	ARdsEventCtrl[314].bSignalInput							:=	NOT bChillerSystemTempHAL; //(* MAIN INC CHILLED WATER *):	 
	ARdsEventCtrl[314].iDelayTimeSV							:=	0;
	ARdsEventCtrl[314].bHoldingDisable;
	ARdsEventCtrl[314].bTest_InvertedInputEn;
	ARdsEventCtrl[314].bEventOutput;
	
	ARdsEventCtrl[315].bSignalInput							:=ARbStnTempPreparationNoRdyAlarm[1];// PROCESS TANK 1 TEMP PREPARATION NO READY ALARM 
	ARdsEventCtrl[315].iDelayTimeSV							:=0;
	ARdsEventCtrl[315].bHoldingDisable;
	ARdsEventCtrl[315].bTest_InvertedInputEn;
	ARdsEventCtrl[315].bEventOutput;

	
	ARdsEventCtrl[316].bSignalInput							:=ARbStnTempPreparationNoRdyAlarm[2];// PROCESS TANK 2 TEMP PREPARATION NO READY ALARM 
	ARdsEventCtrl[316].iDelayTimeSV							:=0;
	ARdsEventCtrl[316].bHoldingDisable;
	ARdsEventCtrl[316].bTest_InvertedInputEn;
	ARdsEventCtrl[316].bEventOutput;

	
	ARdsEventCtrl[317].bSignalInput							:=ARbStnTempPreparationNoRdyAlarm[3];// PROCESS TANK 3 TEMP PREPARATION NO READY ALARM 
	ARdsEventCtrl[317].iDelayTimeSV							:=0;
	ARdsEventCtrl[317].bHoldingDisable;
	ARdsEventCtrl[317].bTest_InvertedInputEn;
	ARdsEventCtrl[317].bEventOutput;

	
	ARdsEventCtrl[318].bSignalInput							:=ARbStnTempPreparationNoRdyAlarm[4];// PROCESS TANK 4 TEMP PREPARATION NO READY ALARM 
	ARdsEventCtrl[318].iDelayTimeSV							:=0;
	ARdsEventCtrl[318].bHoldingDisable;
	ARdsEventCtrl[318].bTest_InvertedInputEn;
	ARdsEventCtrl[318].bEventOutput;

	ARdsEventCtrl[319].bSignalInput							:=ARbStnTempPreparationNoRdyAlarm[5];// PROCESS TANK 5 TEMP PREPARATION NO READY ALARM 
	ARdsEventCtrl[319].iDelayTimeSV							:=0;
	ARdsEventCtrl[319].bHoldingDisable;
	ARdsEventCtrl[319].bTest_InvertedInputEn;
	ARdsEventCtrl[319].bEventOutput;
	
	ARdsEventCtrl[320].bSignalInput							:=ARbStnTempPreparationNoRdyAlarm[6];// PROCESS TANK 6 TEMP PREPARATION NO READY ALARM 
	ARdsEventCtrl[320].iDelayTimeSV							:=0;
	ARdsEventCtrl[320].bHoldingDisable;
	ARdsEventCtrl[320].bTest_InvertedInputEn;
	ARdsEventCtrl[320].bEventOutput;
	
	ARdsEventCtrl[321].bSignalInput							:=ARbStnTempPreparationNoRdyAlarm[7];// PROCESS TANK 7 TEMP PREPARATION NO READY ALARM  
	ARdsEventCtrl[321].iDelayTimeSV							:=0;
	ARdsEventCtrl[321].bHoldingDisable;
	ARdsEventCtrl[321].bTest_InvertedInputEn;
	ARdsEventCtrl[321].bEventOutput;
	
	ARdsEventCtrl[322].bSignalInput							:=ARbStnTempPreparationNoRdyAlarm[8];// PROCESS TANK 8 TEMP PREPARATION NO READY ALARM 
	ARdsEventCtrl[322].iDelayTimeSV							:=0;
	ARdsEventCtrl[322].bHoldingDisable;
	ARdsEventCtrl[322].bTest_InvertedInputEn;
	ARdsEventCtrl[322].bEventOutput;
	
	ARdsEventCtrl[323].bSignalInput							:=FALSE AND ARbStnTempPreparationNoRdyAlarm[9];// PROCESS TANK 9 TEMP PREPARATION NO READY ALARM 
	ARdsEventCtrl[323].iDelayTimeSV							:=0;
	ARdsEventCtrl[323].bHoldingDisable;
	ARdsEventCtrl[323].bTest_InvertedInputEn;
	ARdsEventCtrl[323].bEventOutput;
	
	ARdsEventCtrl[324].bSignalInput							:=ARbStnTempPreparationNoRdyAlarm[10];// PROCESS TANK 10 TEMP PREPARATION NO READY ALARM 
	ARdsEventCtrl[324].iDelayTimeSV							:=0;
	ARdsEventCtrl[324].bHoldingDisable;
	ARdsEventCtrl[324].bTest_InvertedInputEn;
	ARdsEventCtrl[324].bEventOutput;
	
	ARdsEventCtrl[325].bSignalInput							:=FALSE AND ARbStnTempPreparationNoRdyAlarm[11];// PROCESS TANK 11 TEMP PREPARATION NO READY ALARM 
	ARdsEventCtrl[325].iDelayTimeSV							:=0;
	ARdsEventCtrl[325].bHoldingDisable;
	ARdsEventCtrl[325].bTest_InvertedInputEn;
	ARdsEventCtrl[325].bEventOutput;

	
	ARdsEventCtrl[326].bSignalInput							:=FALSE AND ARbStnTempPreparationNoRdyAlarm[12];// PROCESS TANK 12 TEMP PREPARATION NO READY ALARM 
	ARdsEventCtrl[326].iDelayTimeSV							:=0;
	ARdsEventCtrl[326].bHoldingDisable;
	ARdsEventCtrl[326].bTest_InvertedInputEn;
	ARdsEventCtrl[326].bEventOutput;

	
	ARdsEventCtrl[327].bSignalInput							:=FALSE AND bIncTempPreparationNoRdyAlarm;	
	ARdsEventCtrl[327].iDelayTimeSV							:=0;
	ARdsEventCtrl[327].bHoldingDisable;
	ARdsEventCtrl[327].bTest_InvertedInputEn;
	ARdsEventCtrl[327].bEventOutput;

	
	ARdsEventCtrl[328].bSignalInput							:=FALSE AND ARbStnWaterJacketTempPreparationNoRdyAlarm[4];
	ARdsEventCtrl[328].iDelayTimeSV							:=0;
	ARdsEventCtrl[328].bHoldingDisable;
	ARdsEventCtrl[328].bTest_InvertedInputEn;
	ARdsEventCtrl[328].bEventOutput;
	
	ARdsEventCtrl[329].bSignalInput							:=FALSE;
	ARdsEventCtrl[329].iDelayTimeSV							:=0;
	ARdsEventCtrl[329].bHoldingDisable;
	ARdsEventCtrl[329].bTest_InvertedInputEn;
	ARdsEventCtrl[329].bEventOutput;
	
	ARdsEventCtrl[330].bSignalInput							:=	(bAutoStartPb OR ManualPageEnable) AND ARbStnTemp1stLimitAlarm[1] AND NOT ARbStationFunctionBypass[1]; //PROCESS TANK 1 TEMP OVER 1ST LIMIT ALARM
	ARdsEventCtrl[330].iDelayTimeSV							:=	0;
	ARdsEventCtrl[330].bHoldingDisable;
	ARdsEventCtrl[330].bTest_InvertedInputEn;
	ARdsEventCtrl[330].bEventOutput;
	
	ARdsEventCtrl[331].bSignalInput							:=	(bAutoStartPb OR ManualPageEnable) AND ARbStnTemp1stLimitAlarm[2] AND NOT ARbStationFunctionBypass[2]; //PROCESS TANK 2 TEMP OVER 1ST LIMIT ALARM
	ARdsEventCtrl[331].iDelayTimeSV							:=	0;
	ARdsEventCtrl[331].bHoldingDisable;
	ARdsEventCtrl[331].bTest_InvertedInputEn;
	ARdsEventCtrl[331].bEventOutput;
		
	ARdsEventCtrl[332].bSignalInput							:= 	(bAutoStartPb OR ManualPageEnable) AND ARbStnTemp1stLimitAlarm[3] AND NOT ARbStationFunctionBypass[3]; //PROCESS TANK 3 TEMP OVER 1ST LIMIT ALARM
	ARdsEventCtrl[332].iDelayTimeSV							:=	0;
	ARdsEventCtrl[332].bHoldingDisable;
	ARdsEventCtrl[332].bTest_InvertedInputEn;
	ARdsEventCtrl[332].bEventOutput;
		
	ARdsEventCtrl[333].bSignalInput							:=	(bAutoStartPb OR ManualPageEnable) AND ARbStnTemp1stLimitAlarm[4] AND NOT ARbStationFunctionBypass[4]; //PROCESS TANK 4 TEMP OVER 1ST LIMIT ALARM 
	ARdsEventCtrl[333].iDelayTimeSV							:=	0;
	ARdsEventCtrl[333].bHoldingDisable;
	ARdsEventCtrl[333].bTest_InvertedInputEn;
	ARdsEventCtrl[333].bEventOutput;
		
	ARdsEventCtrl[334].bSignalInput							:=	(bAutoStartPb OR ManualPageEnable) AND ARbStnTemp1stLimitAlarm[5] AND NOT ARbStationFunctionBypass[5]; //PROCESS TANK 5 TEMP OVER 1ST LIMIT ALARM
	ARdsEventCtrl[334].iDelayTimeSV							:=	0;
	ARdsEventCtrl[334].bHoldingDisable;
	ARdsEventCtrl[334].bTest_InvertedInputEn;
	ARdsEventCtrl[334].bEventOutput;
	
	ARdsEventCtrl[335].bSignalInput							:=	(bAutoStartPb OR ManualPageEnable) AND ARbStnTemp1stLimitAlarm[6] AND NOT ARbStationFunctionBypass[6]; //PROCESS TANK 6 TEMP OVER 1ST LIMIT ALARM
	ARdsEventCtrl[335].iDelayTimeSV							:=	0;
	ARdsEventCtrl[335].bHoldingDisable;
	ARdsEventCtrl[335].bTest_InvertedInputEn;
	ARdsEventCtrl[335].bEventOutput;
		
	ARdsEventCtrl[336].bSignalInput							:= 	(bAutoStartPb OR ManualPageEnable) AND ARbStnTemp1stLimitAlarm[7] AND NOT ARbStationFunctionBypass[7]; //PROCESS TANK 7 TEMP OVER 1ST LIMIT ALARM
	ARdsEventCtrl[336].iDelayTimeSV							:=	0;
	ARdsEventCtrl[336].bHoldingDisable;
	ARdsEventCtrl[336].bTest_InvertedInputEn;
	ARdsEventCtrl[336].bEventOutput;
		
	ARdsEventCtrl[337].bSignalInput							:=	(bAutoStartPb OR ManualPageEnable) AND ARbStnTemp1stLimitAlarm[8] AND NOT ARbStationFunctionBypass[8]; //PROCESS TANK 8 TEMP OVER 1ST LIMIT ALARM
	ARdsEventCtrl[337].iDelayTimeSV							:=	0;
	ARdsEventCtrl[337].bHoldingDisable;
	ARdsEventCtrl[337].bTest_InvertedInputEn;
	ARdsEventCtrl[337].bEventOutput;
		
	ARdsEventCtrl[338].bSignalInput							:=	FALSE AND (bAutoStartPb OR ManualPageEnable) AND ARbStnTemp1stLimitAlarm[9] AND NOT ARbStationFunctionBypass[9]; //PROCESS TANK 9 TEMP OVER 1ST LIMIT ALARM;
	ARdsEventCtrl[338].iDelayTimeSV							:=	0;
	ARdsEventCtrl[338].bHoldingDisable;
	ARdsEventCtrl[338].bTest_InvertedInputEn;
	ARdsEventCtrl[338].bEventOutput;
	
	ARdsEventCtrl[339].bSignalInput							:=	(bAutoStartPb OR ManualPageEnable) AND DSStnBasketInfo[10].bAvailibility AND ARbStnTemp1stLimitAlarm[10] AND NOT ARbStationFunctionBypass[10]; //PROCESS TANK 10 TEMP OVER 1ST LIMIT ALARM;
	ARdsEventCtrl[339].iDelayTimeSV							:=	0;
	ARdsEventCtrl[339].bHoldingDisable;
	ARdsEventCtrl[339].bTest_InvertedInputEn;
	ARdsEventCtrl[339].bEventOutput;
	
	ARdsEventCtrl[340].bSignalInput							:=	FALSE AND (bAutoStartPb OR ManualPageEnable) AND ARbStnTemp1stLimitAlarm[10] AND NOT ARbStationFunctionBypass[10]; //PROCESS TANK 10 TEMP OVER 1ST LIMIT ALARM
	ARdsEventCtrl[340].iDelayTimeSV							:=	0;
	ARdsEventCtrl[340].bHoldingDisable;
	ARdsEventCtrl[340].bTest_InvertedInputEn;
	ARdsEventCtrl[340].bEventOutput;
	
	ARdsEventCtrl[341].bSignalInput							:=FALSE AND(bAutoStartPb OR ManualPageEnable) AND ARbStnTemp1stLimitAlarm[11] AND NOT ARbStationFunctionBypass[11]; //PROCESS TANK 11 TEMP OVER 1ST LIMIT ALARM
	ARdsEventCtrl[341].iDelayTimeSV							:=0;
	ARdsEventCtrl[341].bHoldingDisable;
	ARdsEventCtrl[341].bTest_InvertedInputEn;
	ARdsEventCtrl[341].bEventOutput;
	
	ARdsEventCtrl[342].bSignalInput							:=FALSE AND(bAutoStartPb OR ManualPageEnable) AND ARbStnTemp1stLimitAlarm[12] AND NOT ARbStationFunctionBypass[12]; //PROCESS TANK 1 TEMP OVER 1ST LIMIT ALARM
	ARdsEventCtrl[342].iDelayTimeSV							:=0;
	ARdsEventCtrl[342].bHoldingDisable;
	ARdsEventCtrl[342].bTest_InvertedInputEn;
	ARdsEventCtrl[342].bEventOutput;
	
	ARdsEventCtrl[343].bSignalInput							:= FALSE AND (bAutoStartPb OR ManualPageEnable) AND bIncTemp1stLimitAlarm; //INC TEMP OVER 1ST LIMIT ALARM 
	ARdsEventCtrl[343].iDelayTimeSV							:=0;
	ARdsEventCtrl[343].bHoldingDisable;
	ARdsEventCtrl[343].bTest_InvertedInputEn;
	ARdsEventCtrl[343].bEventOutput;
	
	ARdsEventCtrl[344].bSignalInput							:= FALSE AND (bAutoStartPb OR ManualPageEnable) AND ARbStnWaterJacketTemp1stLimitAlarm[4]; // STN4 WATER JACKET TEMP OVER 1ST LIMIT ALARM
	ARdsEventCtrl[344].iDelayTimeSV							:=10;
	ARdsEventCtrl[344].bHoldingDisable;
	ARdsEventCtrl[344].bTest_InvertedInputEn;
	ARdsEventCtrl[344].bEventOutput;
	
	ARdsEventCtrl[345].bSignalInput							:=FALSE;
	ARdsEventCtrl[345].iDelayTimeSV							:=0;
	ARdsEventCtrl[345].bHoldingDisable;
	ARdsEventCtrl[345].bTest_InvertedInputEn;
	ARdsEventCtrl[345].bEventOutput;
	
	ARdsEventCtrl[346].bSignalInput							:=(bAutoStartPb OR ManualPageEnable) AND ARbStnTemp2ndLimitAlarm[1]; // PROCESS TANK 1 TEMP OVER 2ND LIMIT ALARM
	ARdsEventCtrl[346].iDelayTimeSV							:=0;
	ARdsEventCtrl[346].bHoldingDisable;
	ARdsEventCtrl[346].bTest_InvertedInputEn;
	ARdsEventCtrl[346].bEventOutput;
	
	ARdsEventCtrl[347].bSignalInput							:=(bAutoStartPb OR ManualPageEnable) AND ARbStnTemp2ndLimitAlarm[2]; // PROCESS TANK 2 TEMP OVER 2ND LIMIT ALARM
	ARdsEventCtrl[347].iDelayTimeSV							:=0;
	ARdsEventCtrl[347].bHoldingDisable;
	ARdsEventCtrl[347].bTest_InvertedInputEn;
	ARdsEventCtrl[347].bEventOutput;
	
	ARdsEventCtrl[348].bSignalInput							:=(bAutoStartPb OR ManualPageEnable) AND ARbStnTemp2ndLimitAlarm[3]; // PROCESS TANK 3 TEMP OVER 2ND LIMIT ALARM
	ARdsEventCtrl[348].iDelayTimeSV							:=0;
	ARdsEventCtrl[348].bHoldingDisable;
	ARdsEventCtrl[348].bTest_InvertedInputEn;
	ARdsEventCtrl[348].bEventOutput;
	
	ARdsEventCtrl[349].bSignalInput							:=(bAutoStartPb OR ManualPageEnable) AND ARbStnTemp2ndLimitAlarm[4]; // PROCESS TANK 4 TEMP OVER 2ND LIMIT ALARM
	ARdsEventCtrl[349].iDelayTimeSV							:=0;
	ARdsEventCtrl[349].bHoldingDisable;
	ARdsEventCtrl[349].bTest_InvertedInputEn;
	ARdsEventCtrl[349].bEventOutput;
	
	ARdsEventCtrl[350].bSignalInput							:=(bAutoStartPb OR ManualPageEnable) AND ARbStnTemp2ndLimitAlarm[5]; // PROCESS TANK 5 TEMP OVER 2ND LIMIT ALARM
	ARdsEventCtrl[350].iDelayTimeSV							:=0;
	ARdsEventCtrl[350].bHoldingDisable;
	ARdsEventCtrl[350].bTest_InvertedInputEn;
	ARdsEventCtrl[350].bEventOutput;
	
	ARdsEventCtrl[351].bSignalInput							:=(bAutoStartPb OR ManualPageEnable) AND ARbStnTemp2ndLimitAlarm[6]; // PROCESS TANK 6 TEMP OVER 2ND LIMIT ALARM
	ARdsEventCtrl[351].iDelayTimeSV							:=0;
	ARdsEventCtrl[351].bHoldingDisable;
	ARdsEventCtrl[351].bTest_InvertedInputEn;
	ARdsEventCtrl[351].bEventOutput;
	
	ARdsEventCtrl[352].bSignalInput							:=(bAutoStartPb OR ManualPageEnable) AND ARbStnTemp2ndLimitAlarm[7]; // PROCESS TANK 7 TEMP OVER 2ND LIMIT ALARM
	ARdsEventCtrl[352].iDelayTimeSV							:=0;
	ARdsEventCtrl[352].bHoldingDisable;
	ARdsEventCtrl[352].bTest_InvertedInputEn;
	ARdsEventCtrl[352].bEventOutput;
	
	ARdsEventCtrl[353].bSignalInput							:=(bAutoStartPb OR ManualPageEnable) AND ARbStnTemp2ndLimitAlarm[8]; // PROCESS TANK 8 TEMP OVER 2ND LIMIT ALARM 
	ARdsEventCtrl[353].iDelayTimeSV							:=0;
	ARdsEventCtrl[353].bHoldingDisable;
	ARdsEventCtrl[353].bTest_InvertedInputEn;
	ARdsEventCtrl[353].bEventOutput;
	
	ARdsEventCtrl[354].bSignalInput							:=(bAutoStartPb OR ManualPageEnable) AND ARbStnTemp2ndLimitAlarm[9]; // PROCESS TANK 9 TEMP OVER 2ND LIMIT ALARM
	ARdsEventCtrl[354].iDelayTimeSV							:=0;
	ARdsEventCtrl[354].bHoldingDisable;
	ARdsEventCtrl[354].bTest_InvertedInputEn;
	ARdsEventCtrl[354].bEventOutput;
	
	ARdsEventCtrl[355].bSignalInput							:=(bAutoStartPb OR ManualPageEnable) AND ARbStnTemp2ndLimitAlarm[10]; // PROCESS TANK 10 TEMP OVER 2ND LIMIT ALARM
	ARdsEventCtrl[355].iDelayTimeSV							:=0;
	ARdsEventCtrl[355].bHoldingDisable;
	ARdsEventCtrl[355].bTest_InvertedInputEn;
	ARdsEventCtrl[355].bEventOutput;
	
	ARdsEventCtrl[356].bSignalInput							:=(bAutoStartPb OR ManualPageEnable) AND ARbStnTemp2ndLimitAlarm[11]; // PROCESS TANK 11 TEMP OVER 2ND LIMIT ALARM
	ARdsEventCtrl[356].iDelayTimeSV							:=0;
	ARdsEventCtrl[356].bHoldingDisable;
	ARdsEventCtrl[356].bTest_InvertedInputEn;
	ARdsEventCtrl[356].bEventOutput;
	
	ARdsEventCtrl[357].bSignalInput							:=(bAutoStartPb OR ManualPageEnable) AND ARbStnTemp2ndLimitAlarm[12]; // PROCESS TANK 12 TEMP OVER 2ND LIMIT ALARM
	ARdsEventCtrl[357].iDelayTimeSV							:=0;
	ARdsEventCtrl[357].bHoldingDisable;
	ARdsEventCtrl[357].bTest_InvertedInputEn;
	ARdsEventCtrl[357].bEventOutput;
	
	ARdsEventCtrl[358].bSignalInput							:=FALSE AND (bAutoStartPb OR ManualPageEnable) AND bIncTemp2ndLimitAlarm; //INC TEMP OVER 2ND LIMIT ALARM
	ARdsEventCtrl[358].iDelayTimeSV							:=0;
	ARdsEventCtrl[358].bHoldingDisable;
	ARdsEventCtrl[358].bTest_InvertedInputEn;
	ARdsEventCtrl[358].bEventOutput;
	
	ARdsEventCtrl[359].bSignalInput							:=FALSE AND (bAutoStartPb OR ManualPageEnable) AND ARbStnWaterJacketTemp2ndLimitAlarm[4]; //STN4 WATER JACKET TEMP OVER 2ND LIMIT ALARM 
	ARdsEventCtrl[359].iDelayTimeSV							:=0;
	ARdsEventCtrl[359].bHoldingDisable;
	ARdsEventCtrl[359].bTest_InvertedInputEn;
	ARdsEventCtrl[359].bEventOutput;
	
	// ANALOG -  OVER 1ST LIMIT ALARM-
	ARdsEventCtrl[360].bSignalInput							:=	bAutoPreparationPb AND NOT ARbConductivityBypass[1] AND ARbStnConductivityLowAlarm[1]; //	PROCESS TANK 1 CONDUCTIVITY OVER 1ST LIMIT ALARM 
	ARdsEventCtrl[360].iDelayTimeSV							:=3;
	ARdsEventCtrl[360].bHoldingDisable;
	ARdsEventCtrl[360].bTest_InvertedInputEn;
	ARdsEventCtrl[360].bEventOutput;
	
	ARdsEventCtrl[361].bSignalInput							:=	bAutoPreparationPb AND NOT ARbConductivityBypass[2] AND ARbStnConductivityLowAlarm[2]; //	PROCESS TANK 2 CONDUCTIVITY OVER 1ST LIMIT ALARM 
	ARdsEventCtrl[361].iDelayTimeSV							:=3;
	ARdsEventCtrl[361].bHoldingDisable;
	ARdsEventCtrl[361].bTest_InvertedInputEn;
	ARdsEventCtrl[361].bEventOutput;
	
	ARdsEventCtrl[362].bSignalInput							:=	bAutoPreparationPb AND NOT ARbConductivityBypass[3] AND ARbStnConductivityLowAlarm[3]; //	PROCESS TANK 3 CONDUCTIVITY OVER 1ST LIMIT ALARM 
	ARdsEventCtrl[362].iDelayTimeSV							:=3;
	ARdsEventCtrl[362].bHoldingDisable;
	ARdsEventCtrl[362].bTest_InvertedInputEn;
	ARdsEventCtrl[362].bEventOutput;
	
	ARdsEventCtrl[363].bSignalInput							:=	bAutoPreparationPb AND NOT ARbConductivityBypass[4] AND ARbStnConductivityLowAlarm[4]; //	PROCESS TANK 4 CONDUCTIVITY OVER 1ST LIMIT ALARM 
	ARdsEventCtrl[363].iDelayTimeSV							:=3;
	ARdsEventCtrl[363].bHoldingDisable;
	ARdsEventCtrl[363].bTest_InvertedInputEn;
	ARdsEventCtrl[363].bEventOutput;
	
	ARdsEventCtrl[364].bSignalInput							:=	bAutoPreparationPb AND NOT ARbConductivityBypass[5] AND ARbStnConductivityLowAlarm[5]; //	PROCESS TANK 5 CONDUCTIVITY OVER 1ST LIMIT ALARM 
	ARdsEventCtrl[364].iDelayTimeSV							:=3;
	ARdsEventCtrl[364].bHoldingDisable;
	ARdsEventCtrl[364].bTest_InvertedInputEn;
	ARdsEventCtrl[364].bEventOutput;
	
	ARdsEventCtrl[365].bSignalInput							:=	bAutoPreparationPb AND NOT ARbConductivityBypass[6] AND ARbStnConductivityLowAlarm[6];
	ARdsEventCtrl[365].iDelayTimeSV							:=3;
	ARdsEventCtrl[365].bHoldingDisable;
	ARdsEventCtrl[365].bTest_InvertedInputEn;
	ARdsEventCtrl[365].bEventOutput;
	
	ARdsEventCtrl[366].bSignalInput							:=	bAutoPreparationPb AND NOT ARbConductivityBypass[7] AND ARbStnConductivityLowAlarm[7];
	ARdsEventCtrl[366].iDelayTimeSV							:=3;
	ARdsEventCtrl[366].bHoldingDisable;
	ARdsEventCtrl[366].bTest_InvertedInputEn;
	ARdsEventCtrl[366].bEventOutput;
	
	ARdsEventCtrl[367].bSignalInput							:=	bAutoPreparationPb AND NOT ARbConductivityBypass[8] AND ARbStnConductivityLowAlarm[8];
	ARdsEventCtrl[367].iDelayTimeSV							:=3;
	ARdsEventCtrl[367].bHoldingDisable;
	ARdsEventCtrl[367].bTest_InvertedInputEn;
	ARdsEventCtrl[367].bEventOutput;
	
	ARdsEventCtrl[368].bSignalInput							:=	ARbDO[eY10107_Stn01ProcessTankPumpOn_Off] AND bAutoPreparationPb AND NOT ARbFilterPressureBypass[1] AND ARbStnFilterPressureLowAlarm[1]; // PROCESS TANK 1 PRESSURE SWITCH  LOW ALARM
	ARdsEventCtrl[368].iDelayTimeSV							:=30;
	ARdsEventCtrl[368].bHoldingDisable;
	ARdsEventCtrl[368].bTest_InvertedInputEn;
	ARdsEventCtrl[368].bEventOutput;
	
	ARdsEventCtrl[369].bSignalInput							:=	ARbDO[eY10108_Stn02ProcessTankPumpOn_Off] AND bAutoPreparationPb AND NOT ARbFilterPressureBypass[2] AND ARbStnFilterPressureLowAlarm[2]; // PROCESS TANK 2 PRESSURE SWITCH  LOW ALARM;
	ARdsEventCtrl[369].iDelayTimeSV							:=30;
	ARdsEventCtrl[369].bHoldingDisable;
	ARdsEventCtrl[369].bTest_InvertedInputEn;
	ARdsEventCtrl[369].bEventOutput;
	
	ARdsEventCtrl[370].bSignalInput							:=	ARbDO[eY10109_Stn03ProcessTankPumpOn_Off] AND bAutoPreparationPb AND NOT ARbFilterPressureBypass[3] AND ARbStnFilterPressureLowAlarm[3]; // PROCESS TANK 3 PRESSURE SWITCH  LOW ALARM
	ARdsEventCtrl[370].iDelayTimeSV							:=30;
	ARdsEventCtrl[370].bHoldingDisable;
	ARdsEventCtrl[370].bTest_InvertedInputEn;
	ARdsEventCtrl[370].bEventOutput;
	
	ARdsEventCtrl[371].bSignalInput							:=	ARbDO[eY10110_Stn04ProcessTankPumpOn_Off] AND bAutoPreparationPb AND NOT ARbFilterPressureBypass[4] AND ARbStnFilterPressureLowAlarm[4]; // PROCESS TANK 4 PRESSURE SWITCH  LOW ALARM
	ARdsEventCtrl[371].iDelayTimeSV							:=30;
	ARdsEventCtrl[371].bHoldingDisable;
	ARdsEventCtrl[371].bTest_InvertedInputEn;
	ARdsEventCtrl[371].bEventOutput;
	
	ARdsEventCtrl[372].bSignalInput							:=	ARbDO[eY10111_Stn05ProcessTankPumpOn_Off] AND bAutoPreparationPb AND NOT ARbFilterPressureBypass[5] AND ARbStnFilterPressureLowAlarm[5]; // PROCESS TANK 5 PRESSURE SWITCH  LOW ALARM
	ARdsEventCtrl[372].iDelayTimeSV							:=30;
	ARdsEventCtrl[372].bHoldingDisable;
	ARdsEventCtrl[372].bTest_InvertedInputEn;
	ARdsEventCtrl[372].bEventOutput;
	
	ARdsEventCtrl[373].bSignalInput							:=	ARbDO[eY10112_Stn06ProcessTankPumpOn_Off] AND bAutoPreparationPb AND NOT ARbFilterPressureBypass[6] AND ARbStnFilterPressureLowAlarm[6]; // PROCESS TANK 6 PRESSURE SWITCH  LOW ALARM
	ARdsEventCtrl[373].iDelayTimeSV							:=30;
	ARdsEventCtrl[373].bHoldingDisable;
	ARdsEventCtrl[373].bTest_InvertedInputEn;
	ARdsEventCtrl[373].bEventOutput;
	
	ARdsEventCtrl[374].bSignalInput							:=	ARbDO[eY10113_Stn07ProcessTankPumpOn_Off] AND bAutoPreparationPb AND NOT ARbFilterPressureBypass[7] AND ARbStnFilterPressureLowAlarm[7]; // PROCESS TANK 7 PRESSURE SWITCH  LOW ALARM
	ARdsEventCtrl[374].iDelayTimeSV							:=30;
	ARdsEventCtrl[374].bHoldingDisable;
	ARdsEventCtrl[374].bTest_InvertedInputEn;
	ARdsEventCtrl[374].bEventOutput;
	
	ARdsEventCtrl[375].bSignalInput							:=	ARbDO[eY10114_Stn08ProcessTankPumpOn_Off] AND bAutoPreparationPb AND NOT ARbFilterPressureBypass[8] AND ARbStnFilterPressureLowAlarm[8]; // PROCESS TANK 8 PRESSURE SWITCH  LOW ALARM; 
	ARdsEventCtrl[375].iDelayTimeSV							:=30;
	ARdsEventCtrl[375].bHoldingDisable;
	ARdsEventCtrl[375].bTest_InvertedInputEn;
	ARdsEventCtrl[375].bEventOutput;
	
	ARdsEventCtrl[376].bSignalInput							:=	ARbDO[eY10211_Stn09ProcessTankPumpOn_Off] AND bAutoPreparationPb AND NOT ARbFilterPressureBypass[9] AND ARbStnFilterPressureLowAlarm[9]; // PROCESS TANK 9 PRESSURE SWITCH  LOW ALARM;
	ARdsEventCtrl[376].iDelayTimeSV							:=30;
	ARdsEventCtrl[376].bHoldingDisable;
	ARdsEventCtrl[376].bTest_InvertedInputEn;
	ARdsEventCtrl[376].bEventOutput;
	
	ARdsEventCtrl[377].bSignalInput							:=	bAutoPreparationPb AND NOT ARbConductivityBypass[9] AND ARbStnConductivityLowAlarm[9];
	ARdsEventCtrl[377].iDelayTimeSV							:=3;
	ARdsEventCtrl[377].bHoldingDisable;
	ARdsEventCtrl[377].bTest_InvertedInputEn;
	ARdsEventCtrl[377].bEventOutput;
	
	ARdsEventCtrl[378].bSignalInput							:=FALSE;
	ARdsEventCtrl[378].iDelayTimeSV							:=0;
	ARdsEventCtrl[378].bHoldingDisable;
	ARdsEventCtrl[378].bTest_InvertedInputEn;
	ARdsEventCtrl[378].bEventOutput;

	ARdsEventCtrl[379].bSignalInput							:=FALSE;
	ARdsEventCtrl[379].iDelayTimeSV							:=0;
	ARdsEventCtrl[379].bHoldingDisable;
	ARdsEventCtrl[379].bTest_InvertedInputEn;
	ARdsEventCtrl[379].bEventOutput;

// ANALOG - OVER 2ND LIMIT ALARM-
	ARdsEventCtrl[380].bSignalInput							:=	bAutoPreparationPb AND NOT ARbConductivityBypass[1] AND ARbStnConductivityHighAlarm[1]; //	PROCESS 1 CONDUCTIVITY OVER 2ND LIMIT ALARM
	ARdsEventCtrl[380].iDelayTimeSV							:=3;
	ARdsEventCtrl[380].bHoldingDisable;
	ARdsEventCtrl[380].bTest_InvertedInputEn;
	ARdsEventCtrl[380].bEventOutput;
	
	ARdsEventCtrl[381].bSignalInput							:=	bAutoPreparationPb AND NOT ARbConductivityBypass[2] AND ARbStnConductivityHighAlarm[2]; //	PROCESS 2 CONDUCTIVITY OVER 2ND LIMIT ALARM
	ARdsEventCtrl[381].iDelayTimeSV							:=3;
	ARdsEventCtrl[381].bHoldingDisable;
	ARdsEventCtrl[381].bTest_InvertedInputEn;
	ARdsEventCtrl[381].bEventOutput;
	
	ARdsEventCtrl[382].bSignalInput							:=	bAutoPreparationPb AND NOT ARbConductivityBypass[3] AND ARbStnConductivityHighAlarm[3]; //	PROCESS 3 CONDUCTIVITY OVER 2ND LIMIT ALARM
	ARdsEventCtrl[382].iDelayTimeSV							:=3;
	ARdsEventCtrl[382].bHoldingDisable;
	ARdsEventCtrl[382].bTest_InvertedInputEn;
	ARdsEventCtrl[382].bEventOutput;
	
	ARdsEventCtrl[383].bSignalInput							:=	bAutoPreparationPb AND NOT ARbConductivityBypass[4] AND ARbStnConductivityHighAlarm[4]; //	PROCESS 4 CONDUCTIVITY OVER 2ND LIMIT ALARM
	ARdsEventCtrl[383].iDelayTimeSV							:=3;
	ARdsEventCtrl[383].bHoldingDisable;
	ARdsEventCtrl[383].bTest_InvertedInputEn;
	ARdsEventCtrl[383].bEventOutput;
	
	ARdsEventCtrl[384].bSignalInput							:=	bAutoPreparationPb AND NOT ARbConductivityBypass[5] AND ARbStnConductivityHighAlarm[5]; //	PROCESS 5 CONDUCTIVITY OVER 2ND LIMIT ALARM;
	ARdsEventCtrl[384].iDelayTimeSV							:=3;
	ARdsEventCtrl[384].bHoldingDisable;
	ARdsEventCtrl[384].bTest_InvertedInputEn;
	ARdsEventCtrl[384].bEventOutput;
	
	ARdsEventCtrl[385].bSignalInput							:=	bAutoPreparationPb AND NOT ARbConductivityBypass[6] AND ARbStnConductivityHighAlarm[6]; //	PROCESS 6 CONDUCTIVITY OVER 2ND LIMIT ALARM;
	ARdsEventCtrl[385].iDelayTimeSV							:=3;
	ARdsEventCtrl[385].bHoldingDisable;
	ARdsEventCtrl[385].bTest_InvertedInputEn;
	ARdsEventCtrl[385].bEventOutput;
	
	ARdsEventCtrl[386].bSignalInput							:=	bAutoPreparationPb AND NOT ARbConductivityBypass[7] AND ARbStnConductivityHighAlarm[7]; //	PROCESS 7 CONDUCTIVITY OVER 2ND LIMIT ALARM;
	ARdsEventCtrl[386].iDelayTimeSV							:=3;
	ARdsEventCtrl[386].bHoldingDisable;
	ARdsEventCtrl[386].bTest_InvertedInputEn;
	ARdsEventCtrl[386].bEventOutput;
	
	ARdsEventCtrl[387].bSignalInput							:=	bAutoPreparationPb AND NOT ARbConductivityBypass[8] AND ARbStnConductivityHighAlarm[8]; //	PROCESS 8 CONDUCTIVITY OVER 2ND LIMIT ALARM;
	ARdsEventCtrl[387].iDelayTimeSV							:=3;
	ARdsEventCtrl[387].bHoldingDisable;
	ARdsEventCtrl[387].bTest_InvertedInputEn;
	ARdsEventCtrl[387].bEventOutput;
	
	ARdsEventCtrl[388].bSignalInput							:=	ARbDO[eY10107_Stn01ProcessTankPumpOn_Off] AND bAutoPreparationPb AND NOT ARbFilterPressureBypass[1] AND ARbStnFilterPressureHighAlarm[1]; // PROCESS TANK 1 PRESSURE SWITCH  A HIGH ALARM
	ARdsEventCtrl[388].iDelayTimeSV							:=30;
	ARdsEventCtrl[388].bHoldingDisable;
	ARdsEventCtrl[388].bTest_InvertedInputEn;
	ARdsEventCtrl[388].bEventOutput;
	
	ARdsEventCtrl[389].bSignalInput							:=	ARbDO[eY10108_Stn02ProcessTankPumpOn_Off] AND bAutoPreparationPb AND NOT ARbFilterPressureBypass[2] AND ARbStnFilterPressureHighAlarm[2]; // PROCESS TANK 2 PRESSURE SWITCH  A HIGH ALARM
	ARdsEventCtrl[388].iDelayTimeSV							:=30;
	ARdsEventCtrl[389].bHoldingDisable;
	ARdsEventCtrl[389].bTest_InvertedInputEn;
	ARdsEventCtrl[389].bEventOutput;
	
	
	ARdsEventCtrl[390].bSignalInput							:=	ARbDO[eY10109_Stn03ProcessTankPumpOn_Off] AND bAutoPreparationPb AND NOT ARbFilterPressureBypass[3] AND ARbStnFilterPressureHighAlarm[3]; // PROCESS TANK 3 PRESSURE SWITCH  A HIGH ALARM
	ARdsEventCtrl[390].iDelayTimeSV							:=30;
	ARdsEventCtrl[390].bHoldingDisable;
	ARdsEventCtrl[390].bTest_InvertedInputEn;
	ARdsEventCtrl[390].bEventOutput;
	
	ARdsEventCtrl[391].bSignalInput							:= 	ARbDO[eY10110_Stn04ProcessTankPumpOn_Off] AND bAutoPreparationPb AND NOT ARbFilterPressureBypass[4] AND ARbStnFilterPressureHighAlarm[4]; // PROCESS TANK 4 PRESSURE SWITCH  A HIGH ALARM
	ARdsEventCtrl[391].iDelayTimeSV							:=30;
	ARdsEventCtrl[391].bHoldingDisable;
	ARdsEventCtrl[391].bTest_InvertedInputEn;
	ARdsEventCtrl[391].bEventOutput;
		
	ARdsEventCtrl[392].bSignalInput							:=	ARbDO[eY10111_Stn05ProcessTankPumpOn_Off] AND bAutoPreparationPb AND NOT ARbFilterPressureBypass[5] AND ARbStnFilterPressureHighAlarm[5]; // PROCESS TANK 5 PRESSURE SWITCH  A HIGH ALARM
	ARdsEventCtrl[392].iDelayTimeSV							:=30;
	ARdsEventCtrl[392].bHoldingDisable;
	ARdsEventCtrl[392].bTest_InvertedInputEn;
	ARdsEventCtrl[392].bEventOutput;
		
	ARdsEventCtrl[393].bSignalInput							:=	ARbDO[eY10112_Stn06ProcessTankPumpOn_Off] AND bAutoPreparationPb AND NOT ARbFilterPressureBypass[6] AND ARbStnFilterPressureHighAlarm[6]; // PROCESS TANK 6 PRESSURE SWITCH  A HIGH ALARM
	ARdsEventCtrl[393].iDelayTimeSV							:=30;
	ARdsEventCtrl[393].bHoldingDisable;
	ARdsEventCtrl[393].bTest_InvertedInputEn;
	ARdsEventCtrl[393].bEventOutput;
		
	ARdsEventCtrl[394].bSignalInput							:=	ARbDO[eY10113_Stn07ProcessTankPumpOn_Off] AND bAutoPreparationPb AND NOT ARbFilterPressureBypass[7] AND ARbStnFilterPressureHighAlarm[7]; // PROCESS TANK 7 PRESSURE SWITCH  A HIGH ALARM
	ARdsEventCtrl[394].iDelayTimeSV							:=30;
	ARdsEventCtrl[394].bHoldingDisable;
	ARdsEventCtrl[394].bTest_InvertedInputEn;
	ARdsEventCtrl[394].bEventOutput;
	
	ARdsEventCtrl[395].bSignalInput							:=	ARbDO[eY10114_Stn08ProcessTankPumpOn_Off] AND bAutoPreparationPb AND NOT ARbFilterPressureBypass[8] AND ARbStnFilterPressureHighAlarm[8]; // PROCESS TANK 8 PRESSURE SWITCH  A HIGH ALARM
	ARdsEventCtrl[395].iDelayTimeSV							:=30;
	ARdsEventCtrl[395].bHoldingDisable;
	ARdsEventCtrl[395].bTest_InvertedInputEn;
	ARdsEventCtrl[395].bEventOutput;
	
	ARdsEventCtrl[396].bSignalInput							:=	ARbDO[eY10211_Stn09ProcessTankPumpOn_Off] AND bAutoPreparationPb AND NOT ARbFilterPressureBypass[9] AND ARbStnFilterPressureHighAlarm[9]; // PROCESS TANK 9 PRESSURE SWITCH  A HIGH ALARM
	ARdsEventCtrl[396].iDelayTimeSV							:=30;
	ARdsEventCtrl[396].bHoldingDisable;
	ARdsEventCtrl[396].bTest_InvertedInputEn;
	ARdsEventCtrl[396].bEventOutput;
		
	ARdsEventCtrl[397].bSignalInput							:=	bAutoPreparationPb AND NOT ARbConductivityBypass[9] AND ARbStnConductivityHighAlarm[9]; //	PROCESS 9 CONDUCTIVITY OVER 2ND LIMIT ALARM;
	ARdsEventCtrl[397].iDelayTimeSV							:=3;
	ARdsEventCtrl[397].bHoldingDisable;
	ARdsEventCtrl[397].bTest_InvertedInputEn;
	ARdsEventCtrl[397].bEventOutput;
		
	ARdsEventCtrl[398].bSignalInput							:=FALSE;
	ARdsEventCtrl[398].iDelayTimeSV							:=0;
	ARdsEventCtrl[398].bHoldingDisable;
	ARdsEventCtrl[398].bTest_InvertedInputEn;
	ARdsEventCtrl[398].bEventOutput;
	
	ARdsEventCtrl[399].bSignalInput							:=FALSE;
	ARdsEventCtrl[399].iDelayTimeSV							:=0;
	ARdsEventCtrl[399].bHoldingDisable;
	ARdsEventCtrl[399].bTest_InvertedInputEn;
	ARdsEventCtrl[399].bEventOutput;
	
	ARdsEventCtrl[400].bSignalInput							:=	PowerOnDelay.Q AND ARbStnAssignBadBskBit[1]; //Process Tank 1 Bad Basket - Over Tolerance Time
	ARdsEventCtrl[400].iDelayTimeSV							:=	0;
	ARdsEventCtrl[400].bHoldingDisable;
	ARdsEventCtrl[400].bTest_InvertedInputEn;
	ARdsEventCtrl[400].bEventOutput;						
	
	ARdsEventCtrl[401].bSignalInput							:=	 PowerOnDelay.Q AND ARbStnAssignBadBskBit[2]; //Process Tank 2 Bad Basket - Over Tolerance Time
	ARdsEventCtrl[401].iDelayTimeSV							:=	0;
	ARdsEventCtrl[401].bHoldingDisable;
	ARdsEventCtrl[401].bTest_InvertedInputEn;
	ARdsEventCtrl[401].bEventOutput;						
	
	ARdsEventCtrl[402].bSignalInput							:=	 PowerOnDelay.Q AND ARbStnAssignBadBskBit[3]; //Process Tank 3 Bad Basket - Over Tolerance Time
	ARdsEventCtrl[402].iDelayTimeSV							:=	0;
	ARdsEventCtrl[402].bHoldingDisable;
	ARdsEventCtrl[402].bTest_InvertedInputEn;
	ARdsEventCtrl[402].bEventOutput;						
	
	ARdsEventCtrl[403].bSignalInput							:=	 PowerOnDelay.Q AND ARbStnAssignBadBskBit[4]; //Process Tank 4 Bad Basket - Over Tolerance Time
	ARdsEventCtrl[403].iDelayTimeSV							:=	0;
	ARdsEventCtrl[403].bHoldingDisable;
	ARdsEventCtrl[403].bTest_InvertedInputEn;
	ARdsEventCtrl[403].bEventOutput;						
	
	ARdsEventCtrl[404].bSignalInput							:=   PowerOnDelay.Q AND ARbStnAssignBadBskBit[5]; //Process Tank 5 Bad Basket - Over Tolerance Time
	ARdsEventCtrl[404].iDelayTimeSV							:=	0;
	ARdsEventCtrl[404].bHoldingDisable;
	ARdsEventCtrl[404].bTest_InvertedInputEn;
	ARdsEventCtrl[404].bEventOutput;						
	
	ARdsEventCtrl[405].bSignalInput							:=  PowerOnDelay.Q AND ARbStnAssignBadBskBit[6]; //Process Tank 6 Bad Basket - Over Tolerance Time	
	ARdsEventCtrl[405].iDelayTimeSV							:=	0;
	ARdsEventCtrl[405].bHoldingDisable;
	ARdsEventCtrl[405].bTest_InvertedInputEn;
	ARdsEventCtrl[405].bEventOutput;						
	
	ARdsEventCtrl[406].bSignalInput							:=  PowerOnDelay.Q AND ARbStnAssignBadBskBit[7]; //Process Tank 7 Bad Basket - Over Tolerance Time	
	ARdsEventCtrl[406].iDelayTimeSV							:=	0;
	ARdsEventCtrl[406].bHoldingDisable;
	ARdsEventCtrl[406].bTest_InvertedInputEn;
	ARdsEventCtrl[406].bEventOutput;						
	
	ARdsEventCtrl[407].bSignalInput							:=PowerOnDelay.Q AND ARbStnAssignBadBskBit[8]; //Process Tank 8 Bad Basket - Over Tolerance Time;	
	ARdsEventCtrl[407].iDelayTimeSV							:=	0;
	ARdsEventCtrl[407].bHoldingDisable;
	ARdsEventCtrl[407].bTest_InvertedInputEn;
	ARdsEventCtrl[407].bEventOutput;						
	
	ARdsEventCtrl[408].bSignalInput							:=PowerOnDelay.Q AND ARbStnAssignBadBskBit[9]; //Process Tank 9 Bad Basket - Over Tolerance Time;
	ARdsEventCtrl[408].iDelayTimeSV							:=0;
	ARdsEventCtrl[408].bHoldingDisable;
	ARdsEventCtrl[408].bTest_InvertedInputEn;
	ARdsEventCtrl[408].bEventOutput;
	
	ARdsEventCtrl[409].bSignalInput							:=PowerOnDelay.Q AND ARbStnAssignBadBskBit[10]; //Process Tank 10 Bad Basket - Over Tolerance Time;
	ARdsEventCtrl[409].iDelayTimeSV							:=0;
	ARdsEventCtrl[409].bHoldingDisable;
	ARdsEventCtrl[409].bTest_InvertedInputEn;
	ARdsEventCtrl[409].bEventOutput;
	
	ARdsEventCtrl[410].bSignalInput							:= FALSE AND PowerOnDelay.Q AND ARbStnAssignBadBskBit[11]; //Process Tank 11 Bad Basket - Over Tolerance Time
	ARdsEventCtrl[410].iDelayTimeSV							:=0;
	ARdsEventCtrl[410].bHoldingDisable;
	ARdsEventCtrl[410].bTest_InvertedInputEn;
	ARdsEventCtrl[410].bEventOutput;
	
	ARdsEventCtrl[411].bSignalInput							:= FALSE AND PowerOnDelay.Q AND ARbStnAssignBadBskBit[12]; //Process Tank 12 Bad Basket - Over Tolerance Time
	ARdsEventCtrl[411].iDelayTimeSV							:=0;
	ARdsEventCtrl[411].bHoldingDisable;
	ARdsEventCtrl[411].bTest_InvertedInputEn;
	ARdsEventCtrl[411].bEventOutput;
	
	ARdsEventCtrl[412].bSignalInput							:= PowerOnDelay.Q AND ARbArmOvertimeError[1]; //Arm 1 Overtime Error
	ARdsEventCtrl[412].iDelayTimeSV							:=0;
	ARdsEventCtrl[412].bHoldingDisable;
	ARdsEventCtrl[412].bTest_InvertedInputEn;
	ARdsEventCtrl[412].bEventOutput;
	
	ARdsEventCtrl[413].bSignalInput							:= FALSE AND PowerOnDelay.Q AND ARbArmOvertimeError[2]; //Arm 2 Overtime Error
	ARdsEventCtrl[413].iDelayTimeSV							:=0;
	ARdsEventCtrl[413].bHoldingDisable;
	ARdsEventCtrl[413].bTest_InvertedInputEn;
	ARdsEventCtrl[413].bEventOutput;
	
	ARdsEventCtrl[414].bSignalInput							:= PowerOnDelay.Q AND ARbArmLifterError[1]; //SLOW PULL Lifter Error
	ARdsEventCtrl[414].iDelayTimeSV							:=0;
	ARdsEventCtrl[414].bHoldingDisable;
	ARdsEventCtrl[414].bTest_InvertedInputEn;
	ARdsEventCtrl[414].bEventOutput;
// Dosing 
	ARdsEventCtrl[415].bSignalInput							:= ARbStnPumpHealthCheckPulseError[1]; //Process Tank 1 Dosing Pump Health A Check Pulse Error
	ARdsEventCtrl[415].iDelayTimeSV							:=0;
	ARdsEventCtrl[415].bHoldingDisable;
	ARdsEventCtrl[415].bTest_InvertedInputEn;
	ARdsEventCtrl[415].bEventOutput;
	
	ARdsEventCtrl[416].bSignalInput							:= ARbStnPumpHealthCheckPulseError[3];//Process Tank 3 Dosing Pump Health A Check Pulse Error
	ARdsEventCtrl[416].iDelayTimeSV							:=0;
	ARdsEventCtrl[416].bHoldingDisable;
	ARdsEventCtrl[416].bTest_InvertedInputEn;
	ARdsEventCtrl[416].bEventOutput;
	
	ARdsEventCtrl[417].bSignalInput							:=ARbStnPumpHealthCheckPulseError[5];//Process Tank 5 Dosing Pump Health A Check Pulse Error
	ARdsEventCtrl[417].iDelayTimeSV							:=0;
	ARdsEventCtrl[417].bHoldingDisable;
	ARdsEventCtrl[417].bTest_InvertedInputEn;
	ARdsEventCtrl[417].bEventOutput;
	
	ARdsEventCtrl[418].bSignalInput							:=FALSE;
	ARdsEventCtrl[418].iDelayTimeSV							:=0;
	ARdsEventCtrl[418].bHoldingDisable;
	ARdsEventCtrl[418].bTest_InvertedInputEn;
	ARdsEventCtrl[418].bEventOutput;

	ARdsEventCtrl[419].bSignalInput							:=FALSE;
	ARdsEventCtrl[419].iDelayTimeSV							:=0;
	ARdsEventCtrl[419].bHoldingDisable;
	ARdsEventCtrl[419].bTest_InvertedInputEn;
	ARdsEventCtrl[419].bEventOutput;
	
	ARdsEventCtrl[420].bSignalInput							:= FALSE;
	ARdsEventCtrl[420].iDelayTimeSV							:=30;
	ARdsEventCtrl[420].bHoldingDisable;
	ARdsEventCtrl[420].bTest_InvertedInputEn;
	ARdsEventCtrl[420].bEventOutput;
	//Vert
	ARdsEventCtrl[421].bSignalInput							:= NOT VertCoERead.bArm1VertUpOT; // Vert UP OT
	ARdsEventCtrl[421].iDelayTimeSV							:=0;
	ARdsEventCtrl[421].bHoldingDisable;
	ARdsEventCtrl[421].bTest_InvertedInputEn;
	ARdsEventCtrl[421].bEventOutput;
	
	ARdsEventCtrl[422].bSignalInput							:= NOT VertCoERead.bArm1VertDownOT; // Vert Down OT
	ARdsEventCtrl[422].iDelayTimeSV							:=0;
	ARdsEventCtrl[422].bHoldingDisable;
	ARdsEventCtrl[422].bTest_InvertedInputEn;
	ARdsEventCtrl[422].bEventOutput;
	
	ARdsEventCtrl[423].bSignalInput							:= NOT VertCoERead.bArm1ErrStop; // Error Stop
	ARdsEventCtrl[423].iDelayTimeSV							:=0;
	ARdsEventCtrl[423].bHoldingDisable;
	ARdsEventCtrl[423].bTest_InvertedInputEn;
	ARdsEventCtrl[423].bEventOutput;
	//Horzt
	ARdsEventCtrl[424].bSignalInput							:= NOT HorzCoERead.bArm1HorzLdOT; // Horz LD OT;
	ARdsEventCtrl[424].iDelayTimeSV							:=0;
	ARdsEventCtrl[424].bHoldingDisable;
	ARdsEventCtrl[424].bTest_InvertedInputEn;
	ARdsEventCtrl[424].bEventOutput;
	
	ARdsEventCtrl[425].bSignalInput							:= NOT HorzCoERead.bArm1HorzUldOT;// Horz Uld OT
	ARdsEventCtrl[425].iDelayTimeSV							:=0;
	ARdsEventCtrl[425].bHoldingDisable;
	ARdsEventCtrl[425].bTest_InvertedInputEn;
	ARdsEventCtrl[425].bEventOutput;
	
	ARdsEventCtrl[426].bSignalInput							:= NOT HorzCoERead.bArm1HorzErrStop;// Horz Error Stop;
	ARdsEventCtrl[426].iDelayTimeSV							:=0;
	ARdsEventCtrl[426].bHoldingDisable;
	ARdsEventCtrl[426].bTest_InvertedInputEn;
	ARdsEventCtrl[426].bEventOutput;
	
	//slowpull
	ARdsEventCtrl[427].bSignalInput							:=NOT SlowpullCoERead.bSlowpullVertUpOT; // Slowpull Vert Up OT
	ARdsEventCtrl[427].iDelayTimeSV							:=0;
	ARdsEventCtrl[427].bHoldingDisable;
	ARdsEventCtrl[427].bTest_InvertedInputEn;
	ARdsEventCtrl[427].bEventOutput;
	
	ARdsEventCtrl[428].bSignalInput							:=NOT SlowpullCoERead.bSlowpullVertDownOT; // Slowpull Vert Down OT;
	ARdsEventCtrl[428].iDelayTimeSV							:=0;
	ARdsEventCtrl[428].bHoldingDisable;
	ARdsEventCtrl[428].bTest_InvertedInputEn;
	ARdsEventCtrl[428].bEventOutput;
	
	ARdsEventCtrl[429].bSignalInput							:=NOT SlowpullCoERead.bSlowpullErrStop; // Slowpull Error stop;
	ARdsEventCtrl[429].iDelayTimeSV							:=0;
	ARdsEventCtrl[429].bHoldingDisable;
	ARdsEventCtrl[429].bTest_InvertedInputEn;
	ARdsEventCtrl[429].bEventOutput;
	
	//UPS
	ARdsEventCtrl[430].bSignalInput							:= FALSE AND bDCPowerUnknownStatusAlarm; //DC Power Unknown Status Alarm 	
	ARdsEventCtrl[430].iDelayTimeSV							:=0;
	ARdsEventCtrl[430].bHoldingDisable;
	ARdsEventCtrl[430].bTest_InvertedInputEn;
	ARdsEventCtrl[430].bEventOutput;
	
	ARdsEventCtrl[431].bSignalInput							:= FALSE AND bUpsCommUnknownStatusAlarm; //	Ups Comm Unknown Status Alarm
	ARdsEventCtrl[431].iDelayTimeSV							:=0;
	ARdsEventCtrl[431].bHoldingDisable;
	ARdsEventCtrl[431].bTest_InvertedInputEn;
	ARdsEventCtrl[431].bEventOutput;
		
	ARdsEventCtrl[432].bSignalInput							:=bBatteryReplacementRequestAlarm; //Battery Replacement Request Alarm 
	ARdsEventCtrl[432].iDelayTimeSV							:=0;
	ARdsEventCtrl[432].bHoldingDisable;
	ARdsEventCtrl[432].bTest_InvertedInputEn;
	ARdsEventCtrl[432].bEventOutput;
		
	ARdsEventCtrl[433].bSignalInput							:=bUpsCommErrorAlarm; //Ups Comm Error Alarm
	ARdsEventCtrl[433].iDelayTimeSV							:=0;
	ARdsEventCtrl[433].bHoldingDisable;
	ARdsEventCtrl[433].bTest_InvertedInputEn;
	ARdsEventCtrl[433].bEventOutput;
		
	ARdsEventCtrl[434].bSignalInput							:=DSArm1VertConfig.MC_ArmError; //Arm 1 Vertical Axis Error 
	ARdsEventCtrl[434].iDelayTimeSV							:=0;
	ARdsEventCtrl[434].bHoldingDisable;
	ARdsEventCtrl[434].bTest_InvertedInputEn;
	ARdsEventCtrl[434].bEventOutput;
	
	ARdsEventCtrl[435].bSignalInput							:=DSArm1HorzConfig.MC_ArmError; //Arm 1 Horizontal Axis Error
	ARdsEventCtrl[435].iDelayTimeSV							:=0;
	ARdsEventCtrl[435].bHoldingDisable;
	ARdsEventCtrl[435].bTest_InvertedInputEn;
	ARdsEventCtrl[435].bEventOutput;
		
	ARdsEventCtrl[436].bSignalInput							:=DSArm2VertConfig.MC_ArmError; //Arm 2 Vertical Axis Error 
	ARdsEventCtrl[436].iDelayTimeSV							:=0;
	ARdsEventCtrl[436].bHoldingDisable;
	ARdsEventCtrl[436].bTest_InvertedInputEn;
	ARdsEventCtrl[436].bEventOutput;
		
	ARdsEventCtrl[437].bSignalInput							:=DSArm2HorzConfig.MC_ArmError; //Arm 2 Horizontal Axis Error
	ARdsEventCtrl[437].iDelayTimeSV							:=0;
	ARdsEventCtrl[437].bHoldingDisable;
	ARdsEventCtrl[437].bTest_InvertedInputEn;
	ARdsEventCtrl[437].bEventOutput;
		
//	MasterTimeBlock 
	ARdsEventCtrl[438].bSignalInput							:=bMTBWriteArmDataError; //Master Time Block Write Arm Data Error 
	ARdsEventCtrl[438].iDelayTimeSV							:=0;
	ARdsEventCtrl[438].bHoldingDisable;
	ARdsEventCtrl[438].bTest_InvertedInputEn;
	ARdsEventCtrl[438].bEventOutput;
	
	ARdsEventCtrl[439].bSignalInput							:=bMTBWriteStnDataError; //Master Time Block Write Stn Data Error
	ARdsEventCtrl[439].iDelayTimeSV							:=0;
	ARdsEventCtrl[439].bHoldingDisable;
	ARdsEventCtrl[439].bTest_InvertedInputEn;
	ARdsEventCtrl[439].bEventOutput;
	
	ARdsEventCtrl[440].bSignalInput							:= bMTBNoAvailableSlotError; //	Master Time Block No Available Slot Error
	ARdsEventCtrl[440].iDelayTimeSV							:=0; 
	ARdsEventCtrl[440].bHoldingDisable;
	ARdsEventCtrl[440].bTest_InvertedInputEn;
	ARdsEventCtrl[440].bEventOutput;
	
	ARdsEventCtrl[441].bSignalInput							:= FALSE; //	
	ARdsEventCtrl[441].iDelayTimeSV							:=3;
	ARdsEventCtrl[441].bHoldingDisable;
	ARdsEventCtrl[441].bTest_InvertedInputEn;
	ARdsEventCtrl[441].bEventOutput;
	
	ARdsEventCtrl[442].bSignalInput							:=FALSE; 
	ARdsEventCtrl[442].iDelayTimeSV							:=0;
	ARdsEventCtrl[442].bHoldingDisable;
	ARdsEventCtrl[442].bTest_InvertedInputEn;
	ARdsEventCtrl[442].bEventOutput;
	
	ARdsEventCtrl[443].bSignalInput							:=FALSE; 
	ARdsEventCtrl[443].iDelayTimeSV							:=0;
	ARdsEventCtrl[443].bHoldingDisable;
	ARdsEventCtrl[443].bTest_InvertedInputEn;
	ARdsEventCtrl[443].bEventOutput;
	
//ProductRecipe	
	ARdsEventCtrl[444].bSignalInput							:=DSfbGnrProductRecipeMemoryOut.bCallArmSpeedProfileMemoryErr AND ARbProductRecipeCallEn[0]; //Loading Call Arm Speed Profile Memory Error
	ARdsEventCtrl[444].iDelayTimeSV							:=0;
	ARdsEventCtrl[444].bHoldingDisable;
	ARdsEventCtrl[444].bTest_InvertedInputEn;
	ARdsEventCtrl[444].bEventOutput;
	
	ARdsEventCtrl[445].bSignalInput							:=DSfbGnrProductRecipeMemoryOut.bCallPickStationNoErr AND ARbProductRecipeCallEn[0]; //Loading Call Pick Station No Error
	ARdsEventCtrl[445].iDelayTimeSV							:=0;
	ARdsEventCtrl[445].bHoldingDisable;
	ARdsEventCtrl[445].bTest_InvertedInputEn;
	ARdsEventCtrl[445].bEventOutput;
	
	ARdsEventCtrl[446].bSignalInput							:=DSfbGnrProductRecipeMemoryOut.bCallTransferStationNoErr AND ARbProductRecipeCallEn[0]; //Loading Call Transfer Station No Error
	ARdsEventCtrl[446].iDelayTimeSV							:=0;
	ARdsEventCtrl[446].bHoldingDisable;
	ARdsEventCtrl[446].bTest_InvertedInputEn;
	ARdsEventCtrl[446].bEventOutput;
	
	ARdsEventCtrl[447].bSignalInput							:=DSfbGnrProductRecipeMemoryOut.bCallUpDownPatternMemoryErr AND ARbProductRecipeCallEn[0]; //Loading Call Up Down Pattern Memory Error
	ARdsEventCtrl[447].iDelayTimeSV							:=0;
	ARdsEventCtrl[447].bHoldingDisable;
	ARdsEventCtrl[447].bTest_InvertedInputEn;
	ARdsEventCtrl[447].bEventOutput;
	
	ARdsEventCtrl[448].bSignalInput							:=DSfbGnrProductRecipeMemoryOut.bInvalidProductRecipeNoErrHold AND ARbProductRecipeCallEn[0]; //Loading Invalid Product Recipe No Error Hold
	ARdsEventCtrl[448].iDelayTimeSV							:=0;
	ARdsEventCtrl[448].bHoldingDisable;
	ARdsEventCtrl[448].bTest_InvertedInputEn;
	ARdsEventCtrl[448].bEventOutput;
	
	ARdsEventCtrl[449].bSignalInput							:=DSfbGnrProductRecipeMemoryOut.bInvalidProductRecipeStepErrHold AND ARbProductRecipeCallEn[0]; //Loading Invalid Product Recipe Step Error Hold
	ARdsEventCtrl[449].iDelayTimeSV							:=0;
	ARdsEventCtrl[449].bHoldingDisable;
	ARdsEventCtrl[449].bTest_InvertedInputEn;
	ARdsEventCtrl[449].bEventOutput;
	
	ARdsEventCtrl[450].bSignalInput							:= DSfbGnrProductRecipeMemoryOut.bCallArmSpeedProfileMemoryErr AND 
											(ARbProductRecipeCallEn[1] OR
											 ARbProductRecipeCallEn[2] OR
											 ARbProductRecipeCallEn[3] OR
											 ARbProductRecipeCallEn[4] OR
											 ARbProductRecipeCallEn[5] OR
											 ARbProductRecipeCallEn[6] OR
											 ARbProductRecipeCallEn[7] OR
											 ARbProductRecipeCallEn[8] OR
											 ARbProductRecipeCallEn[9] OR
											 ARbProductRecipeCallEn[10] OR
											 ARbProductRecipeCallEn[11] OR
											 ARbProductRecipeCallEn[12]) ; //Station Call Arm Speed Profile Memory Error
	ARdsEventCtrl[450].iDelayTimeSV							:=3;
	ARdsEventCtrl[450].bHoldingDisable;
	ARdsEventCtrl[450].bTest_InvertedInputEn;
	ARdsEventCtrl[450].bEventOutput;
	
	ARdsEventCtrl[451].bSignalInput							:= DSfbGnrProductRecipeMemoryOut.bCallPickStationNoErr AND
											(ARbProductRecipeCallEn[1] OR
											 ARbProductRecipeCallEn[2] OR
											 ARbProductRecipeCallEn[3] OR
											 ARbProductRecipeCallEn[4] OR
											 ARbProductRecipeCallEn[5] OR
											 ARbProductRecipeCallEn[6] OR
 											 ARbProductRecipeCallEn[7] OR
											 ARbProductRecipeCallEn[8] OR
											 ARbProductRecipeCallEn[9] OR
											 ARbProductRecipeCallEn[10] OR
											 ARbProductRecipeCallEn[11] OR
											 ARbProductRecipeCallEn[12]) ; // Station Call Pick Station No Error
	ARdsEventCtrl[451].iDelayTimeSV							:=3;
	ARdsEventCtrl[451].bHoldingDisable;
	ARdsEventCtrl[451].bTest_InvertedInputEn;
	ARdsEventCtrl[451].bEventOutput;
	
	ARdsEventCtrl[452].bSignalInput							:=DSfbGnrProductRecipeMemoryOut.bCallTransferStationNoErr AND
											(ARbProductRecipeCallEn[1] OR
											 ARbProductRecipeCallEn[2] OR
											 ARbProductRecipeCallEn[3] OR
											 ARbProductRecipeCallEn[4] OR
											 ARbProductRecipeCallEn[5] OR
											 ARbProductRecipeCallEn[6] OR
											 ARbProductRecipeCallEn[7] OR
											 ARbProductRecipeCallEn[8] OR
											 ARbProductRecipeCallEn[9] OR
											 ARbProductRecipeCallEn[10] OR
											 ARbProductRecipeCallEn[11] OR
											 ARbProductRecipeCallEn[12]); //Station Call Transfer Station No Error								 											  
	ARdsEventCtrl[452].iDelayTimeSV							:=0;
	ARdsEventCtrl[452].bHoldingDisable;
	ARdsEventCtrl[452].bTest_InvertedInputEn;
	ARdsEventCtrl[452].bEventOutput;
	
	ARdsEventCtrl[453].bSignalInput							:= DSfbGnrProductRecipeMemoryOut.bCallUpDownPatternMemoryErr AND
											(ARbProductRecipeCallEn[1] OR
											 ARbProductRecipeCallEn[2] OR
											 ARbProductRecipeCallEn[3] OR
											 ARbProductRecipeCallEn[4] OR
											 ARbProductRecipeCallEn[5] OR
											 ARbProductRecipeCallEn[6] OR
 											 ARbProductRecipeCallEn[7] OR
											 ARbProductRecipeCallEn[8] OR
											 ARbProductRecipeCallEn[9] OR
											 ARbProductRecipeCallEn[10] OR
											 ARbProductRecipeCallEn[11] OR
											 ARbProductRecipeCallEn[12]); //Station Call Up Down Pattern Memory Error
	ARdsEventCtrl[453].iDelayTimeSV							:=0;
	ARdsEventCtrl[453].bHoldingDisable;
	ARdsEventCtrl[453].bTest_InvertedInputEn;
	ARdsEventCtrl[453].bEventOutput;
	
	ARdsEventCtrl[454].bSignalInput							:= DSfbGnrProductRecipeMemoryOut.bInvalidProductRecipeNoErrHold AND
											(ARbProductRecipeCallEn[1] OR
											 ARbProductRecipeCallEn[2] OR
											 ARbProductRecipeCallEn[3] OR
											 ARbProductRecipeCallEn[4] OR
											 ARbProductRecipeCallEn[5] OR
											 ARbProductRecipeCallEn[6] OR
 											 ARbProductRecipeCallEn[7] OR
											 ARbProductRecipeCallEn[8] OR
											 ARbProductRecipeCallEn[9] OR
											 ARbProductRecipeCallEn[10] OR
											 ARbProductRecipeCallEn[11] OR
											 ARbProductRecipeCallEn[12]); // Station Invalid Product Recipe No Error Hold
	ARdsEventCtrl[454].iDelayTimeSV							:=0;
	ARdsEventCtrl[454].bHoldingDisable;
	ARdsEventCtrl[454].bTest_InvertedInputEn;
	ARdsEventCtrl[454].bEventOutput;
	
	ARdsEventCtrl[455].bSignalInput							:=DSfbGnrProductRecipeMemoryOut.bInvalidProductRecipeStepErrHold AND
											(ARbProductRecipeCallEn[1] OR
											 ARbProductRecipeCallEn[2] OR
											 ARbProductRecipeCallEn[3] OR
											 ARbProductRecipeCallEn[4] OR
											 ARbProductRecipeCallEn[5] OR
											 ARbProductRecipeCallEn[6] OR
 											 ARbProductRecipeCallEn[7] OR
											 ARbProductRecipeCallEn[8] OR
											 ARbProductRecipeCallEn[9] OR
											 ARbProductRecipeCallEn[10] OR
											 ARbProductRecipeCallEn[11] OR
											 ARbProductRecipeCallEn[12]); //Station Invalid Product Recipe Step Error Hold
	ARdsEventCtrl[455].iDelayTimeSV							:=0;
	ARdsEventCtrl[455].bHoldingDisable;
	ARdsEventCtrl[455].bTest_InvertedInputEn;
	ARdsEventCtrl[455].bEventOutput;
	
	ARdsEventCtrl[456].bSignalInput							:=FALSE;
	ARdsEventCtrl[456].iDelayTimeSV							:=0;
	ARdsEventCtrl[456].bHoldingDisable;
	ARdsEventCtrl[456].bTest_InvertedInputEn;
	ARdsEventCtrl[456].bEventOutput;
	
	ARdsEventCtrl[457].bSignalInput							:=FALSE;
	ARdsEventCtrl[457].iDelayTimeSV							:=0;
	ARdsEventCtrl[457].bHoldingDisable;
	ARdsEventCtrl[457].bTest_InvertedInputEn;
	ARdsEventCtrl[457].bEventOutput;
	
	ARdsEventCtrl[458].bSignalInput							:=FALSE;
	ARdsEventCtrl[458].iDelayTimeSV							:=0;
	ARdsEventCtrl[458].bHoldingDisable;
	ARdsEventCtrl[458].bTest_InvertedInputEn;
	ARdsEventCtrl[458].bEventOutput;
	
	ARdsEventCtrl[459].bSignalInput							:=FALSE;
	ARdsEventCtrl[459].iDelayTimeSV							:=0;
	ARdsEventCtrl[459].bHoldingDisable;
	ARdsEventCtrl[459].bTest_InvertedInputEn;
	ARdsEventCtrl[459].bEventOutput;
	
	ARdsEventCtrl[460].bSignalInput							:= FALSE; 
	ARdsEventCtrl[460].iDelayTimeSV							:=3;
	ARdsEventCtrl[460].bHoldingDisable;
	ARdsEventCtrl[460].bTest_InvertedInputEn;
	ARdsEventCtrl[460].bEventOutput;
	
	ARdsEventCtrl[461].bSignalInput							:= FALSE; 
	ARdsEventCtrl[461].iDelayTimeSV							:=3;
	ARdsEventCtrl[461].bHoldingDisable;
	ARdsEventCtrl[461].bTest_InvertedInputEn;
	ARdsEventCtrl[462].bSignalInput							:=FALSE; 
	ARdsEventCtrl[461].bEventOutput;
	
	ARdsEventCtrl[462].iDelayTimeSV							:=0;
	ARdsEventCtrl[462].bHoldingDisable;
	ARdsEventCtrl[462].bTest_InvertedInputEn;
	ARdsEventCtrl[462].bEventOutput;
	
	ARdsEventCtrl[463].bSignalInput							:=FALSE; 
	ARdsEventCtrl[463].iDelayTimeSV							:=0;
	ARdsEventCtrl[463].bHoldingDisable;
	ARdsEventCtrl[463].bTest_InvertedInputEn;
	ARdsEventCtrl[463].bEventOutput;
	
	ARdsEventCtrl[464].bSignalInput							:=FALSE; 
	ARdsEventCtrl[464].iDelayTimeSV							:=0;
	ARdsEventCtrl[464].bHoldingDisable;
	ARdsEventCtrl[464].bTest_InvertedInputEn;
	ARdsEventCtrl[464].bEventOutput;
	
	ARdsEventCtrl[465].bSignalInput							:=FALSE;
	ARdsEventCtrl[465].iDelayTimeSV							:=0;
	ARdsEventCtrl[465].bHoldingDisable;
	ARdsEventCtrl[465].bTest_InvertedInputEn;
	ARdsEventCtrl[465].bEventOutput;
	
	ARdsEventCtrl[466].bSignalInput							:=FALSE;
	ARdsEventCtrl[466].iDelayTimeSV							:=0;
	ARdsEventCtrl[466].bHoldingDisable;
	ARdsEventCtrl[466].bTest_InvertedInputEn;
	ARdsEventCtrl[466].bEventOutput;
	
	ARdsEventCtrl[467].bSignalInput							:=FALSE;
	ARdsEventCtrl[467].iDelayTimeSV							:=0;
	ARdsEventCtrl[467].bHoldingDisable;
	ARdsEventCtrl[467].bTest_InvertedInputEn;
	ARdsEventCtrl[467].bEventOutput;
	
	ARdsEventCtrl[468].bSignalInput							:=FALSE;
	ARdsEventCtrl[468].iDelayTimeSV							:=0;
	ARdsEventCtrl[468].bHoldingDisable;
	ARdsEventCtrl[468].bTest_InvertedInputEn;
	ARdsEventCtrl[468].bEventOutput;
	
	ARdsEventCtrl[469].bSignalInput							:=FALSE;
	ARdsEventCtrl[469].iDelayTimeSV							:=0;
	ARdsEventCtrl[469].bHoldingDisable;
	ARdsEventCtrl[469].bTest_InvertedInputEn;
	ARdsEventCtrl[469].bEventOutput;
	
	ARdsEventCtrl[470].bSignalInput							:=FALSE; 
	ARdsEventCtrl[470].iDelayTimeSV							:=0;
	ARdsEventCtrl[470].bHoldingDisable;
	ARdsEventCtrl[470].bTest_InvertedInputEn;
	ARdsEventCtrl[470].bEventOutput;
	
	ARdsEventCtrl[471].bSignalInput							:=FALSE;  
	ARdsEventCtrl[471].iDelayTimeSV							:=0;
	ARdsEventCtrl[471].bHoldingDisable;
	ARdsEventCtrl[471].bTest_InvertedInputEn;
	ARdsEventCtrl[471].bEventOutput;
	
	ARdsEventCtrl[472].bSignalInput							:=FALSE; 
	ARdsEventCtrl[472].iDelayTimeSV							:=0;
	ARdsEventCtrl[472].bHoldingDisable;
	ARdsEventCtrl[472].bTest_InvertedInputEn;
	ARdsEventCtrl[472].bEventOutput;
	
	ARdsEventCtrl[473].bSignalInput							:=FALSE; 
	ARdsEventCtrl[473].iDelayTimeSV							:=0;
	ARdsEventCtrl[473].bHoldingDisable;
	ARdsEventCtrl[473].bTest_InvertedInputEn;
	ARdsEventCtrl[473].bEventOutput;
	
	ARdsEventCtrl[474].bSignalInput							:=FALSE; 
	ARdsEventCtrl[474].iDelayTimeSV							:=0;
	ARdsEventCtrl[474].bHoldingDisable;
	ARdsEventCtrl[474].bTest_InvertedInputEn;
	ARdsEventCtrl[474].bEventOutput;
	
	ARdsEventCtrl[475].bSignalInput							:=FALSE; 
	ARdsEventCtrl[475].iDelayTimeSV							:=0;
	ARdsEventCtrl[475].bHoldingDisable;
	ARdsEventCtrl[475].bTest_InvertedInputEn;
	ARdsEventCtrl[475].bEventOutput;
	
	ARdsEventCtrl[476].bSignalInput							:=FALSE;
	ARdsEventCtrl[476].iDelayTimeSV							:=0;
	ARdsEventCtrl[476].bHoldingDisable;
	ARdsEventCtrl[476].bTest_InvertedInputEn;
	ARdsEventCtrl[476].bEventOutput;
	
	ARdsEventCtrl[477].bSignalInput							:=FALSE;
	ARdsEventCtrl[477].iDelayTimeSV							:=0;
	ARdsEventCtrl[477].bHoldingDisable;
	ARdsEventCtrl[477].bTest_InvertedInputEn;
	ARdsEventCtrl[477].bEventOutput;
	
	ARdsEventCtrl[478].bSignalInput							:=FALSE;
	ARdsEventCtrl[478].iDelayTimeSV							:=0;
	ARdsEventCtrl[478].bHoldingDisable;
	ARdsEventCtrl[478].bTest_InvertedInputEn;
	ARdsEventCtrl[478].bEventOutput;

	ARdsEventCtrl[479].bSignalInput							:=FALSE;
	ARdsEventCtrl[479].iDelayTimeSV							:=0;
	ARdsEventCtrl[479].bHoldingDisable;
	ARdsEventCtrl[479].bTest_InvertedInputEn;
	ARdsEventCtrl[479].bEventOutput;

	ARdsEventCtrl[480].bSignalInput							:=FALSE; 
	ARdsEventCtrl[480].iDelayTimeSV							:=0;
	ARdsEventCtrl[480].bHoldingDisable;
	ARdsEventCtrl[480].bTest_InvertedInputEn;
	ARdsEventCtrl[480].bEventOutput;
	
	ARdsEventCtrl[481].bSignalInput							:=FALSE;
	ARdsEventCtrl[481].iDelayTimeSV							:=0;
	ARdsEventCtrl[481].bHoldingDisable;
	ARdsEventCtrl[481].bTest_InvertedInputEn;
	ARdsEventCtrl[481].bEventOutput;
	
	ARdsEventCtrl[482].bSignalInput							:=FALSE; 
	ARdsEventCtrl[482].iDelayTimeSV							:=0;
	ARdsEventCtrl[482].bHoldingDisable;
	ARdsEventCtrl[482].bTest_InvertedInputEn;
	ARdsEventCtrl[482].bEventOutput;
	
	ARdsEventCtrl[483].bSignalInput							:=FALSE; 
	ARdsEventCtrl[483].iDelayTimeSV							:=0;
	ARdsEventCtrl[483].bHoldingDisable;
	ARdsEventCtrl[483].bTest_InvertedInputEn;
	ARdsEventCtrl[483].bEventOutput;
	
	ARdsEventCtrl[484].bSignalInput							:=FALSE;
	ARdsEventCtrl[484].iDelayTimeSV							:=0;
	ARdsEventCtrl[484].bHoldingDisable;
	ARdsEventCtrl[484].bTest_InvertedInputEn;
	ARdsEventCtrl[484].bEventOutput;
	
	ARdsEventCtrl[485].bSignalInput							:=FALSE;
	ARdsEventCtrl[485].iDelayTimeSV							:=0;
	ARdsEventCtrl[485].bHoldingDisable;
	ARdsEventCtrl[485].bTest_InvertedInputEn;
	ARdsEventCtrl[485].bEventOutput;
	
	ARdsEventCtrl[486].bSignalInput							:=FALSE;
	ARdsEventCtrl[486].iDelayTimeSV							:=0;
	ARdsEventCtrl[486].bHoldingDisable;
	ARdsEventCtrl[486].bTest_InvertedInputEn;
	ARdsEventCtrl[486].bEventOutput;
	
	ARdsEventCtrl[487].bSignalInput							:=FALSE;
	ARdsEventCtrl[487].iDelayTimeSV							:=0;
	ARdsEventCtrl[487].bHoldingDisable;
	ARdsEventCtrl[487].bTest_InvertedInputEn;
	ARdsEventCtrl[487].bEventOutput;
	
	ARdsEventCtrl[488].bSignalInput							:=FALSE;
	ARdsEventCtrl[488].iDelayTimeSV							:=0;
	ARdsEventCtrl[488].bHoldingDisable;
	ARdsEventCtrl[488].bTest_InvertedInputEn;
	ARdsEventCtrl[488].bEventOutput;
	
	ARdsEventCtrl[489].bSignalInput							:=FALSE;
	ARdsEventCtrl[489].iDelayTimeSV							:=0;
	ARdsEventCtrl[489].bHoldingDisable;
	ARdsEventCtrl[489].bTest_InvertedInputEn;
	ARdsEventCtrl[489].bEventOutput;
	
	ARdsEventCtrl[490].bSignalInput							:=FALSE; 
	ARdsEventCtrl[490].iDelayTimeSV							:=0;
	ARdsEventCtrl[490].bHoldingDisable;
	ARdsEventCtrl[490].bTest_InvertedInputEn;
	ARdsEventCtrl[490].bEventOutput;
	
	
	ARdsEventCtrl[491].bSignalInput							:=FALSE; 
	ARdsEventCtrl[491].iDelayTimeSV							:=0;
	ARdsEventCtrl[491].bHoldingDisable;
	ARdsEventCtrl[491].bTest_InvertedInputEn;
	ARdsEventCtrl[491].bEventOutput;
	
		
	ARdsEventCtrl[492].bSignalInput							:=FALSE; 
	ARdsEventCtrl[492].iDelayTimeSV							:=0;
	ARdsEventCtrl[492].bHoldingDisable;
	ARdsEventCtrl[492].bTest_InvertedInputEn;
	ARdsEventCtrl[492].bEventOutput;
	
		
	ARdsEventCtrl[493].bSignalInput							:=FALSE; 
	ARdsEventCtrl[493].iDelayTimeSV							:=0;
	ARdsEventCtrl[493].bHoldingDisable;
	ARdsEventCtrl[493].bTest_InvertedInputEn;
	ARdsEventCtrl[493].bEventOutput;
	
	ARdsEventCtrl[494].bSignalInput							:=FALSE; 
	ARdsEventCtrl[494].iDelayTimeSV							:=0;
	ARdsEventCtrl[494].bHoldingDisable;
	ARdsEventCtrl[494].bTest_InvertedInputEn;
	ARdsEventCtrl[494].bEventOutput;
	
	
	ARdsEventCtrl[495].bSignalInput							:=FALSE; 
	ARdsEventCtrl[495].iDelayTimeSV							:=0;
	ARdsEventCtrl[495].bHoldingDisable;
	ARdsEventCtrl[495].bTest_InvertedInputEn;
	ARdsEventCtrl[495].bEventOutput;
	
	
	ARdsEventCtrl[496].bSignalInput							:=FALSE;
	ARdsEventCtrl[496].iDelayTimeSV							:=0;
	ARdsEventCtrl[496].bHoldingDisable;
	ARdsEventCtrl[496].bTest_InvertedInputEn;
	ARdsEventCtrl[496].bEventOutput;
	
		
	ARdsEventCtrl[497].bSignalInput							:=FALSE;
	ARdsEventCtrl[497].iDelayTimeSV							:=0;
	ARdsEventCtrl[497].bHoldingDisable;
	ARdsEventCtrl[497].bTest_InvertedInputEn;
	ARdsEventCtrl[497].bEventOutput;
	
		
	ARdsEventCtrl[498].bSignalInput							:= FALSE ;
	ARdsEventCtrl[498].iDelayTimeSV							:=0;
	ARdsEventCtrl[498].bHoldingDisable						:=TRUE;	
	ARdsEventCtrl[498].bTest_InvertedInputEn;
	ARdsEventCtrl[498].bEventOutput;
	
	
	ARdsEventCtrl[499].bSignalInput							:=FALSE;
	ARdsEventCtrl[499].iDelayTimeSV							:=0;
	ARdsEventCtrl[499].bHoldingDisable						:=TRUE;
	ARdsEventCtrl[499].bTest_InvertedInputEn;
	ARdsEventCtrl[499].bEventOutput;
	
	
	ARdsEventCtrl[500].bSignalInput							:=FALSE;
	ARdsEventCtrl[500].iDelayTimeSV							:=0;
	ARdsEventCtrl[500].bHoldingDisable						:=TRUE;
	ARdsEventCtrl[500].bTest_InvertedInputEn;
	ARdsEventCtrl[500].bEventOutput;

END_PROGRAM

// ---- POUs/MainProgram/AlertCtrl/MisshookSensorCtrl.TcPOU
PROGRAM MisshookSensorCtrl
VAR

	bArm1LdMisshookDetectZone			: BOOL;
	ARbArm1StnMisshookDetectZone		: ARRAY [1..iStnQty] OF BOOL;
	bArm1UldMisshookDetectZone			: BOOL;

	bArm1DeactDetectZone				: BOOL;

END_VAR

(*ARM 1*)
(******Misshook 1 Alarm Control*******)

IF PowerOnDelay.Q AND (bAutoStartPb OR ManualPageEnable ) AND NOT ARbArmMissHookByPass1[1]
AND
(
(
( ARDSArmCtrl[1].AR3sbPositionCfm[2,1,1] OR (NOT ARDSArmCtrl[1].AR3sbPositionCfm[2,1,1] AND bArm1MisshookDetectZone))
AND
DSArmBasketInfo[1].bAvailibility AND NOT ARbMAP_ArmMisshookSensorA[1])
OR
(NOT DSArmBasketInfo[1].bAvailibility AND bArm1MisshookDetectZone AND ARbMAP_ArmMisshookSensorA[1])
)
THEN

ARbArmMisshook1Alarm[1] := TRUE;
ELSE
ARbArmMisshook1Alarm[1] := FALSE;

END_IF

(******Misshook 2 Alarm Control*******)

IF PowerOnDelay.Q AND (bAutoStartPb OR ManualPageEnable ) AND NOT ARbArmMissHookByPass2[1]
AND
(
(
( ARDSArmCtrl[1].AR3sbPositionCfm[2,1,1] OR (NOT ARDSArmCtrl[1].AR3sbPositionCfm[2,1,1] AND bArm1MisshookDetectZone))
AND
DSArmBasketInfo[1].bAvailibility AND NOT ARbMAP_ArmMisshookSensorA[2]
)
OR
(NOT DSArmBasketInfo[1].bAvailibility AND bArm1MisshookDetectZone AND ARbMAP_ArmMisshookSensorA[2])
)
THEN

ARbArmMisshook2Alarm[1] := TRUE;
ELSE
ARbArmMisshook2Alarm[1] := FALSE;

END_IF

(*
(******Misshook 1 Alarm Control*******)                       	(********************* Funtion for Arm that have two baskets on it *********************)

IF PowerOnDelay.Q AND (bAutoStartPb OR ManualPageEnable ) AND NOT ARbArmMissHookByPass1[1]
AND
(
(
( ARDSArmCtrl[1].AR3sbPositionCfm[2,1,1] OR (NOT ARDSArmCtrl[1].AR3sbPositionCfm[2,1,1] AND bArm1MisshookDetectZone))
AND
((DSArmBasketInfo[1].bAvailibility_A AND NOT X116_10) OR (DSArmBasketInfo[1].bAvailibility_B AND NOT X116_12))
)
OR
(NOT DSArmBasketInfo[1].bAvailibility AND bArm1MisshookDetectZone AND (X116_10 OR X116_12)  )
)
THEN

ARbArmMisshook1Alarm[1] := TRUE;
ELSE
ARbArmMisshook1Alarm[1] := FALSE;

END_IF

(******Misshook 2 Alarm Control*******)			(********************* Funtion for Arm that have two baskets on it *********************)

IF PowerOnDelay.Q AND (bAutoStartPb OR ManualPageEnable ) AND NOT ARbArmMissHookByPass2[1]
AND
(
(
( ARDSArmCtrl[1].AR3sbPositionCfm[2,1,1] OR (NOT ARDSArmCtrl[1].AR3sbPositionCfm[2,1,1] AND bArm1MisshookDetectZone))
AND
((DSArmBasketInfo[1].bAvailibility_A AND NOT X116_11) OR (DSArmBasketInfo[1].bAvailibility_B AND NOT X116_13))
)
OR
(NOT DSArmBasketInfo[1].bAvailibility AND bArm1MisshookDetectZone AND (X116_11 OR X116_13)  )
)
THEN

ARbArmMisshook2Alarm[1] := TRUE;
ELSE
ARbArmMisshook2Alarm[1] := FALSE;

END_IF
*)


(*Arm 1*)

IF ARbLdHorzZoneConfirm[1] AND (*ARlrVertPositionMM[1]*)DSArm1VertConfig.lrGen_Out_CurrentPos < ( ARDSArmCtrl[1].AR3slrPosition[2,1,6] - ARlrArmDetectZoneRange[1]) THEN
bArm1LdMisshookDetectZone := TRUE;
ELSE
bArm1LdMisshookDetectZone := FALSE;
END_IF

IF ARbArm1HorzStnZoneConfirm[1]  AND (*ARlrVertPositionMM[1]*)DSArm1VertConfig.lrGen_Out_CurrentPos < ( ARDSArmCtrl[1].AR3slrPosition[1,1,6] - ARlrArmDetectZoneRange[1]) THEN
ARbArm1StnMisshookDetectZone[1] := TRUE;
ELSE
ARbArm1StnMisshookDetectZone[1] := FALSE;
END_IF

IF ARbArm1HorzStnZoneConfirm[2]  AND DSArm1VertConfig.lrGen_Out_CurrentPos < ( ARDSArmCtrl[1].AR3slrPosition[1,2,6] - ARlrArmDetectZoneRange[2]) THEN
ARbArm1StnMisshookDetectZone[2] := TRUE;
ELSE
ARbArm1StnMisshookDetectZone[2] := FALSE;
END_IF

IF ARbArm1HorzStnZoneConfirm[3]  AND DSArm1VertConfig.lrGen_Out_CurrentPos < ( ARDSArmCtrl[1].AR3slrPosition[1,3,6] - ARlrArmDetectZoneRange[3]) THEN
ARbArm1StnMisshookDetectZone[3] := TRUE;
ELSE
ARbArm1StnMisshookDetectZone[3] := FALSE;
END_IF

IF ARbArm1HorzStnZoneConfirm[4]  AND DSArm1VertConfig.lrGen_Out_CurrentPos < ( ARDSArmCtrl[1].AR3slrPosition[1,4,6] - ARlrArmDetectZoneRange[4]) THEN
ARbArm1StnMisshookDetectZone[4] := TRUE;
ELSE
ARbArm1StnMisshookDetectZone[4] := FALSE;
END_IF

IF ARbArm1HorzStnZoneConfirm[5]  AND DSArm1VertConfig.lrGen_Out_CurrentPos < ( ARDSArmCtrl[1].AR3slrPosition[1,5,6] - ARlrArmDetectZoneRange[5]) THEN
ARbArm1StnMisshookDetectZone[5] := TRUE;
ELSE
ARbArm1StnMisshookDetectZone[5] := FALSE;
END_IF

IF ARbArm1HorzStnZoneConfirm[6]  AND DSArm1VertConfig.lrGen_Out_CurrentPos < ( ARDSArmCtrl[1].AR3slrPosition[1,6,6] - ARlrArmDetectZoneRange[6]) THEN
ARbArm1StnMisshookDetectZone[6] := TRUE;
ELSE
ARbArm1StnMisshookDetectZone[6] := FALSE;
END_IF

IF ARbArm1HorzStnZoneConfirm[7]  AND DSArm1VertConfig.lrGen_Out_CurrentPos < ( ARDSArmCtrl[1].AR3slrPosition[1,7,6] - ARlrArmDetectZoneRange[7]) THEN
ARbArm1StnMisshookDetectZone[7] := TRUE;
ELSE
ARbArm1StnMisshookDetectZone[7] := FALSE;
END_IF

IF ARbArm1HorzStnZoneConfirm[8]  AND DSArm1VertConfig.lrGen_Out_CurrentPos < ( ARDSArmCtrl[1].AR3slrPosition[1,8,6] - ARlrArmDetectZoneRange[8]) THEN
ARbArm1StnMisshookDetectZone[8] := TRUE;
ELSE
ARbArm1StnMisshookDetectZone[8] := FALSE;
END_IF

// STN 9 with slowpull
IF ARbArm1HorzStnZoneConfirm[9]  AND 
(
(NOT DSArmBasketInfo[1].bAvailibility AND DSArm1VertConfig.lrGen_Out_CurrentPos < ( ARDSArmCtrl[1].AR3slrPosition[1,9,6] - ARlrArmStnDetectZoneRange[1,9])) 
OR
(DSArmBasketInfo[1].bAvailibility AND DSArm1VertConfig.lrGen_Out_CurrentPos < ( ARDSArmCtrl[1].AR3slrPosition[1,9,2] - ARlrArmDetectZoneRange[9]))
)
THEN
ARbArm1StnMisshookDetectZone[9] := TRUE;
ELSE
ARbArm1StnMisshookDetectZone[9] := FALSE;
END_IF

IF ARbArm1HorzStnZoneConfirm[10]  AND DSArm1VertConfig.lrGen_Out_CurrentPos < ( ARDSArmCtrl[1].AR3slrPosition[1,10,6] - ARlrArmDetectZoneRange[10]) THEN
ARbArm1StnMisshookDetectZone[10] := TRUE;
ELSE
ARbArm1StnMisshookDetectZone[10] := FALSE;
END_IF

IF ARbArm1HorzStnZoneConfirm[11]  AND DSArm1VertConfig.lrGen_Out_CurrentPos < ( ARDSArmCtrl[1].AR3slrPosition[1,11,6] - ARlrArmDetectZoneRange[11]) THEN
ARbArm1StnMisshookDetectZone[11] := TRUE;
ELSE
ARbArm1StnMisshookDetectZone[11] := FALSE;
END_IF

IF ARbArm1HorzStnZoneConfirm[12]  AND DSArm1VertConfig.lrGen_Out_CurrentPos < ( ARDSArmCtrl[1].AR3slrPosition[1,12,6] - ARlrArmDetectZoneRange[12]) THEN
ARbArm1StnMisshookDetectZone[12] := TRUE;
ELSE
ARbArm1StnMisshookDetectZone[12] := FALSE;
END_IF


IF ARbUldHorzZoneConfirm[1] AND DSArm1VertConfig.lrGen_Out_CurrentPos < ( ARDSArmCtrl[1].AR3slrPosition[3,1,6] - ARlrArmDetectZoneRange[1]) THEN
bArm1UldMisshookDetectZone := TRUE;
ELSE
bArm1UldMisshookDetectZone := FALSE;
END_IF

(*
IF ARbArm1HorzStnZoneConfirm[6]  AND
(
(NOT DSArmBasketInfo[1].bAvailibility AND DSArm1VertConfig.lrGen_Out_CurrentPos < ( ARDSArmCtrl[1].AR3slrPosition[1,6,6] - ARlrArmStnDetectZoneRange[1,6]))
OR
( DSArmBasketInfo[1].bAvailibility AND DSArm1VertConfig.lrGen_Out_CurrentPos < ( ARDSArmCtrl[1].AR3slrPosition[1,6,2] - ARlrArmDetectZoneRange[6] (*ARlrArmStnDetectZoneRange[1,6]*)))
)
THEN
ARbArm1StnMisshookDetectZone[6] := TRUE;
ELSE
ARbArm1StnMisshookDetectZone[6] := FALSE;
END_IF
*)


IF DSArm1VertConfig.lrGen_Out_CurrentPos > INT_TO_LREAL( ARiArmDeactDetectZoneRange[1]) THEN
bArm1DeactDetectZone := TRUE;
ELSE
bArm1DeactDetectZone := FALSE;
END_IF


IF ARbArmVertHomeDone[1] AND ARbArmHorzHomeDone[1] AND NOT bArm1DeactDetectZone THEN

	IF ARDSArmCtrl[1].AR3sbPositionCfm[2,1,1] THEN
	bArm1MisshookDetectZone:= TRUE;

	ELSIF bArm1LdMisshookDetectZone THEN
	bArm1MisshookDetectZone:= TRUE;

	ELSIF ARbArm1StnMisshookDetectZone[1] THEN
	bArm1MisshookDetectZone:= TRUE;

	ELSIF ARbArm1StnMisshookDetectZone[2] THEN
	bArm1MisshookDetectZone:= TRUE;

	ELSIF ARbArm1StnMisshookDetectZone[3] THEN
	bArm1MisshookDetectZone:= TRUE;

	ELSIF ARbArm1StnMisshookDetectZone[4] THEN
	bArm1MisshookDetectZone:= TRUE;

	ELSIF ARbArm1StnMisshookDetectZone[5] THEN
	bArm1MisshookDetectZone:= TRUE;

	ELSIF ARbArm1StnMisshookDetectZone[6] THEN
	bArm1MisshookDetectZone:= TRUE;

	ELSIF ARbArm1StnMisshookDetectZone[7] THEN
	bArm1MisshookDetectZone:= TRUE;

	ELSIF ARbArm1StnMisshookDetectZone[8] THEN
	bArm1MisshookDetectZone:= TRUE;

	ELSIF ARbArm1StnMisshookDetectZone[9] THEN
	bArm1MisshookDetectZone:= TRUE;

	ELSIF ARbArm1StnMisshookDetectZone[10] THEN
	bArm1MisshookDetectZone:= TRUE;

	ELSIF ARbArm1StnMisshookDetectZone[11] THEN
	bArm1MisshookDetectZone:= TRUE;

	ELSIF ARbArm1StnMisshookDetectZone[12] THEN
	bArm1MisshookDetectZone:= TRUE;

	ELSIF bArm1UldMisshookDetectZone THEN
	bArm1MisshookDetectZone:= TRUE;

	ELSE
	bArm1MisshookDetectZone:= FALSE;
	END_IF

ELSE
bArm1MisshookDetectZone:= FALSE;

END_IF

END_PROGRAM

// ---- POUs/MainProgram/AlertCtrl/DeactivateCtrl.TcPOU
PROGRAM DeactivateCtrl
VAR
	ARbDeactivateTestPB : ARRAY [1..iDeactivateQty] OF BOOL;
END_VAR

// ARdsEventCtrl[250] - ARdsEventCtrl[298]

(*xxxxxxxxxxxx Deactivate xxxxxxxxxx*)
   
  ARdsEventCtrl[250].bSignalInput :=ARbDeactivated[eY10100_Stn01UltrasonicGeneratorLeftRightOnOff];	//STN 01 ULTRASONIC GENERATOR ON/OFF (-10U1)     
  ARdsEventCtrl[251].bSignalInput :=DE10101;	//STN 02 ULTRASONIC GENERATOR ON/OFF (-11U1)     
  ARdsEventCtrl[252].bSignalInput :=DE10102;	//STN 04 ULTRASONIC GENERATOR ON/OFF (-12U1)     
  ARdsEventCtrl[253].bSignalInput :=DE10103;	//STN 05 ULTRASONIC GENERATOR ON/OFF (-13U1)     
  ARdsEventCtrl[254].bSignalInput :=DE10104;	//STN 07 ULTRASONIC GENERATOR ON/OFF (-14U1)     
  ARdsEventCtrl[255].bSignalInput :=DE10105;	//STN 08 ULTRASONIC GENERATOR ON/OFF (-15U1)     
  ARdsEventCtrl[256].bSignalInput :=DE10106;	//STN 07 DI WATER RETURN TANK PUMP ON/OFF (-81K1)
  ARdsEventCtrl[257].bSignalInput :=DE10107;	//STN 01 PROCESS TANK PUMP ON/OFF (-73K1)        
  ARdsEventCtrl[258].bSignalInput :=DE10108;	//STN 02 PROCESS TANK PUMP ON/OFF (-74K1)        
  ARdsEventCtrl[259].bSignalInput :=DE10109;	//STN 03 PROCESS TANK PUMP ON/OFF (-75K1)        
  ARdsEventCtrl[260].bSignalInput :=DE10110;	//STN 04 PROCESS TANK PUMP ON/OFF (-76K1)        
  ARdsEventCtrl[261].bSignalInput :=DE10111;	//STN 05 PROCESS TANK PUMP ON/OFF (-77K1)   
  ARdsEventCtrl[262].bSignalInput :=DE10112;	//STN 06 PROCESS TANK PUMP ON/OFF (-78K1)   
  ARdsEventCtrl[263].bSignalInput :=DE10113;	//STN 07 PROCESS TANK PUMP ON/OFF (-79K1)   
  ARdsEventCtrl[264].bSignalInput :=DE10114;	//STN 08 PROCESS TANK PUMP ON/OFF (-80K1)   
  ARdsEventCtrl[265].bSignalInput :=DE10115;	//STN 01 PROCESS TANK HEATER ON/OFF (-130K1)
  ARdsEventCtrl[266].bSignalInput :=DE10200;	//STN 02 PROCESS TANK HEATER ON/OFF (-131K1) 
  ARdsEventCtrl[267].bSignalInput :=DE10201;	//STN 03 PROCESS TANK HEATER ON/OFF (-132K1) 
  ARdsEventCtrl[268].bSignalInput :=DE10202;	//STN 04 PROCESS TANK HEATER ON/OFF (-133K1) 
  ARdsEventCtrl[269].bSignalInput :=DE10203;	//STN 05 PROCESS TANK HEATER ON/OFF (-134K1) 
  ARdsEventCtrl[270].bSignalInput :=DE10204;	//STN 06 PROCESS TANK HEATER ON/OFF (-135K1) 
  ARdsEventCtrl[271].bSignalInput :=DE10205;	//STN 07 PROCESS TANK HEATER ON/OFF (-136K1)
  ARdsEventCtrl[272].bSignalInput :=DE10206;	//STN 08 PROCESS TANK HEATER ON/OFF (-137K1) 
  ARdsEventCtrl[273].bSignalInput :=DE10207;	//STN 10 PROCESS TANK HEATER ON/OFF (-138K1) 
  ARdsEventCtrl[274].bSignalInput :=DE10208;	//STN 09 - STN 10 FFU UNIT ON/OFF (-163K1)   
  ARdsEventCtrl[275].bSignalInput :=DE10209;	//UNLOADING FFU UNIT ON/OFF (-164K1)         
  ARdsEventCtrl[276].bSignalInput :=DE10210;	//UNLOADING CONVEYOR FFU UNIT ON/OFF (-165K1)
  ARdsEventCtrl[277].bSignalInput :=DE10211;	//STN 09 PROCESS TANK PUMP ON/OFF (-82K1)    
  ARdsEventCtrl[278].bSignalInput :=DE10300;	//STN 01 - 08 AGITATION MOTOR ON/OFF (-160K1)                                   
  ARdsEventCtrl[279].bSignalInput :=DE10301;	//LOADING CONVEYOR 01 ON/OFF (-170K1)                                           
  ARdsEventCtrl[280].bSignalInput :=DE10302;	//LOADING CONVEYOR 02 ON/OFF (-171K1)                                           
  ARdsEventCtrl[281].bSignalInput :=DE10303;	//LOADING CONVEYOR 03 ON/OFF (-172K1)                                           
  ARdsEventCtrl[282].bSignalInput :=DE10304;	//LOADING CONVEYOR 04 ON/OFF (-173K1)
  ARdsEventCtrl[283].bSignalInput :=DE10305;	//UNLOADING CONVEYOR 01 ON/OFF (-174K1)
  ARdsEventCtrl[284].bSignalInput :=DE10306;	//UNLOADING CONVEYOR 02 ON/OFF (-175K1)
  ARdsEventCtrl[285].bSignalInput :=DE10307;	//UNLOADING CONVEYOR 03 ON/OFF (-176K1)
  ARdsEventCtrl[286].bSignalInput :=DE10308;	//UNLOADING CONVEYOR 04 ON/OFF (-177K1)
  ARdsEventCtrl[287].bSignalInput :=DE11100;	//STN 03 MEGASONIC GENERATOR 01 ON/OFF (-16U1))      
  ARdsEventCtrl[288].bSignalInput :=DE11101;	//STN 03 MEGASONIC GENERATOR 02 ON/OFF (-17U1))      
  ARdsEventCtrl[289].bSignalInput :=DE11102;	//STN 01 DOSING PUMP ON/OFF (-70K1)               
  ARdsEventCtrl[290].bSignalInput :=DE11103;	//STN 03 DOSING PUMP ON/OFF (-71K1)  
  ARdsEventCtrl[291].bSignalInput :=DE12000;	//STN 03 DOSING PUMP ON/OFF (-71K1)              
  ARdsEventCtrl[292].bSignalInput :=DE12001;	//STN 05 DOSING PUMP ON/OFF (-72K1)           
  ARdsEventCtrl[293].bSignalInput :=DE12002;	//STN 06 MEGASONIC GENERATOR 01 ON/OFF (-18U1)
  ARdsEventCtrl[294].bSignalInput :=DE12003;	//STN 06 MEGASONIC GENERATOR 02 ON/OFF (-19U1)
  ARdsEventCtrl[295].bSignalInput :=DE12004;	//STN 06 MEGASONIC GENERATOR 03 ON/OFF (-20U1) 
  ARdsEventCtrl[296].bSignalInput :=ARbArmMissHookByPass1[1];	
  ARdsEventCtrl[297].bSignalInput :=ARbArmMissHookByPass2[1];	
  ARdsEventCtrl[298].bSignalInput :=ARwDO[eY11003_GeneralBuzzerTone02].00;	
(*
(********************************************************************************** DEACTIVATED - ( ARbDeactivateOutput[1] - ARbDeactivateOutput[16] )**********************************************************************************)
(*Deactivate*)
ARsDeactivateDescription	[1]		:=		'[ DA-0001 ] OutputSignal - DEACTIVATED Reserved ';
ARbDeactivateOutput		[1]		:=		FALSE OR ARbDeactivateTestPB[1];

(*Deactivate*)
ARsDeactivateDescription	[2]		:=		'[ DA-0002 ] OutputSignal - Reserved';
ARbDeactivateOutput		[2]		:=		FALSE OR ARbDeactivateTestPB[2];

(*Deactivate*)
ARsDeactivateDescription	[3]		:=		'[ DA-0003 ] OutputSignal - Reserved';
ARbDeactivateOutput		[3]		:=		FALSE OR ARbDeactivateTestPB[3];

(*Deactivate*)
ARsDeactivateDescription	[4]		:=		'[ DA-0004 ] OutputSignal - Reserved';
ARbDeactivateOutput		[4]		:=		FALSE OR ARbDeactivateTestPB[4];

(*Deactivate*)
ARsDeactivateDescription	[5]		:=		'[ DA-0005 ] OutputSignal - Reserved';
ARbDeactivateOutput		[5]		:=		FALSE OR ARbDeactivateTestPB[5];

(*Deactivate*)
ARsDeactivateDescription	[6]		:=		'[ DA-0006 ] OutputSignal - Reserved';
ARbDeactivateOutput		[6]		:=		FALSE OR ARbDeactivateTestPB[6];

(*Deactivate*)
ARsDeactivateDescription	[7]		:=		'[ DA-0007 ] OutputSignal - Reserved';
ARbDeactivateOutput		[7]		:=		FALSE OR ARbDeactivateTestPB[7];

(*Deactivate*)
ARsDeactivateDescription	[8]		:=		'[ DA-0008 ] OutputSignal - Reserved';
ARbDeactivateOutput		[8]		:=		FALSE OR ARbDeactivateTestPB[8];

(*Deactivate*)
ARsDeactivateDescription	[9]		:=		'[ DA-0009 ] OutputSignal - Reserved ';
ARbDeactivateOutput		[9]		:=		FALSE OR ARbDeactivateTestPB[9];

(*Deactivate*)
ARsDeactivateDescription	[10]		:=		'[ DA-0010 ] OutputSignal - Reserved ';
ARbDeactivateOutput		[10]		:=		FALSE OR ARbDeactivateTestPB[10];

(*Deactivate*)
ARsDeactivateDescription	[11]		:=		'[ DA-0011 ] OutputSignal - Reserved ';
ARbDeactivateOutput		[11]		:=		FALSE OR ARbDeactivateTestPB[11];

(*Deactivate*)
ARsDeactivateDescription	[12]		:=		'[ DA-0012 ] OutputSignal - Reserved ';
ARbDeactivateOutput		[12]		:=		FALSE OR ARbDeactivateTestPB[12];

(*Deactivate*)
ARsDeactivateDescription	[13]		:=		'[ DA-0013 ] OutputSignal - Reserved ';
ARbDeactivateOutput		[13]		:=		FALSE OR ARbDeactivateTestPB[13];

(*Deactivate*)
ARsDeactivateDescription	[14]		:=		'[ DA-0014 ] OutputSignal - Reserved ';
ARbDeactivateOutput		[14]		:=		FALSE OR ARbDeactivateTestPB[14];

(*Deactivate*)
ARsDeactivateDescription	[15]		:=		'[ DA-0015 ] OutputSignal - Reserved';
ARbDeactivateOutput		[15]		:=		FALSE OR ARbDeactivateTestPB[15];

(*Deactivate*)
ARsDeactivateDescription	[16]		:=		'[ DA-0016 ] OutputSignal - Reserved';
ARbDeactivateOutput		[16]		:=		FALSE OR ARbDeactivateTestPB[16];

(********************************************************************************** DEACTIVATED - ( ARbDeactivateOutput[17] - ARbDeactivateOutput[32] )**********************************************************************************)

(*Deactivate*)
ARsDeactivateDescription	[17]		:=		'[ DA-0017 ] OutputSignal - DEACTIVATED STN 1 PROCESS TANK PUMP ON/OFF (-50K1) ';
ARbDeactivateOutput		[17]		:=		DE10100 OR ARbDeactivateTestPB[17];

(*Deactivate*)
ARsDeactivateDescription	[18]		:=		'[ DA-0018 ] OutputSignal - DEACTIVATED STN 2 PROCESS TANK PUMP ON/OFF (-51K1) ';
ARbDeactivateOutput		[18]		:=		DE10101 OR ARbDeactivateTestPB[18];

(*Deactivate*)
ARsDeactivateDescription	[19]		:=		'[ DA-0019 ] OutputSignal - DEACTIVATED STN 3 PROCESS TANK PUMP ON/OFF (-52K1) ';
ARbDeactivateOutput		[19]		:=		DE10102 OR ARbDeactivateTestPB[19];

(*Deactivate*)
ARsDeactivateDescription	[20]		:=		'[ DA-0020 ] OutputSignal - DEACTIVATED STN 5 VACUUM PUMP ON/OFF (-56K1) ';
ARbDeactivateOutput		[20]		:=		DE10103 OR ARbDeactivateTestPB[20];

(*Deactivate*)
ARsDeactivateDescription	[21]		:=		'[ DA-0021 ] OutputSignal - DEACTIVATED STN 2&3 AGITATION MOTOR ON/OFF (-25K1) ';
ARbDeactivateOutput		[21]		:=		DE10104 OR ARbDeactivateTestPB[21];

(*Deactivate*)
ARsDeactivateDescription	[22]		:=		'[ DA-0022 ] OutputSignal - DEACTIVATED STN 5 BLOWER ON/OFF (-65K1) ';
ARbDeactivateOutput		[22]		:=		DE10105 OR ARbDeactivateTestPB[22];

(*Deactivate*)
ARsDeactivateDescription	[23]		:=		'[ DA-0023 ] OutputSignal - DEACTIVATED STN 1 SUB PROCESS TANK STIRRING MOTOR ON/OFF (-26K1) ';
ARbDeactivateOutput		[23]		:=		DE10106 OR ARbDeactivateTestPB[23];

(*Deactivate*)
ARsDeactivateDescription	[24]		:=		'[ DA-0024 ] OutputSignal - DEACTIVATED DETERGENT TANK 1 STIRRING MOTOR ON/OFF (-27K1) ';
ARbDeactivateOutput		[24]		:=		DE10107 OR ARbDeactivateTestPB[24];

(*Deactivate*)
ARsDeactivateDescription	[25]		:=		'[ DA-0025 ] OutputSignal - DEACTIVATED STN 1 ULTRASONIC ON/OFF (-16K1) ';
ARbDeactivateOutput		[25]		:=		DE10108 OR ARbDeactivateTestPB[25];

(*Deactivate*)
ARsDeactivateDescription	[26]		:=		'[ DA-0026 ] OutputSignal - DEACTIVATED STN 2 ULTRASONIC ON/OFF (-17K1) ';
ARbDeactivateOutput		[26]		:=		DE10109 OR ARbDeactivateTestPB[26];

(*Deactivate*)
ARsDeactivateDescription	[27]		:=		'[ DA-0027 ] OutputSignal - DEACTIVATED STN 3 ULTRASONIC ON/OFF (-18K1) ';
ARbDeactivateOutput		[27]		:=		DE10110 OR ARbDeactivateTestPB[27];

(*Deactivate*)
ARsDeactivateDescription	[28]		:=		'[ DA-0028 ] OutputSignal - DEACTIVATED STN 1 ELECTRIC ACTUATOR ON/OFF (-21K1) ';
ARbDeactivateOutput		[28]		:=		DE10111 OR ARbDeactivateTestPB[28];

(*Deactivate*)
ARsDeactivateDescription	[29]		:=		'[ DA-0029 ] OutputSignal - DEACTIVATED STN 2 ELECTRIC ACTUATOR ON/OFF (-22K1) ';
ARbDeactivateOutput		[29]		:=		DE10112 OR ARbDeactivateTestPB[29];

(*Deactivate*)
ARsDeactivateDescription	[30]		:=		'[ DA-0030 ] OutputSignal - DEACTIVATED STN 3 ELECTRIC ACTUATOR ON/OFF (-23K1)  ';
ARbDeactivateOutput		[30]		:=		DE10113 OR ARbDeactivateTestPB[30];

(*Deactivate*)
ARsDeactivateDescription	[31]		:=		'[ DA-0031 ] OutputSignal - DEACTIVATED RESERVED ';
ARbDeactivateOutput		[31]		:=		DE10114 OR ARbDeactivateTestPB[31];

(*Deactivate*)
ARsDeactivateDescription	[32]		:=		'[ DA-0032 ] OutputSignal - DEACTIVATED RESERVED ';
ARbDeactivateOutput		[32]		:=		DE10115 OR ARbDeactivateTestPB[32];

(********************************************************************************** DEACTIVATED - ( ARbDeactivateOutput[33] - ARbDeactivateOutput[48] )**********************************************************************************)

(*Deactivate*)
ARsDeactivateDescription	[33]		:=		'[ DA-0033 ] OutputSignal - DEACTIVATED STN 5 PROCESS TANK HEATER A ON/OFF (-70K1) ';
ARbDeactivateOutput		[33]		:=		DE10200 OR ARbDeactivateTestPB[33];

(*Deactivate*)
ARsDeactivateDescription	[34]		:=		'[ DA-0034 ] OutputSignal - DEACTIVATED STN 5 PROCESS TANK HEATER B ON/OFF (-71K1) ';
ARbDeactivateOutput		[34]		:=		DE10201 OR ARbDeactivateTestPB[34];

(*Deactivate*)
ARsDeactivateDescription	[35]		:=		'[ DA-0035 ] OutputSignal - DEACTIVATED STN 1 SUB PROCESS TANK HEATER ON/OFF (-72K1) ';
ARbDeactivateOutput		[35]		:=		DE10202 OR ARbDeactivateTestPB[35];

(*Deactivate*)
ARsDeactivateDescription	[36]		:=		'[ DA-0036 ] OutputSignal - DEACTIVATED STN 2 SUB PROCESS TANK HEATER ON/OFF (-73K1) ';
ARbDeactivateOutput		[36]		:=		DE10203 OR ARbDeactivateTestPB[36];

(*Deactivate*)
ARsDeactivateDescription	[37]		:=		'[ DA-0037 ] OutputSignal - DEACTIVATED STN 3 SUB PROCESS TANK HEATER ON/OFF (-74K1) ';
ARbDeactivateOutput		[37]		:=		DE10204 OR ARbDeactivateTestPB[37];

(*Deactivate*)
ARsDeactivateDescription	[38]		:=		'[ DA-0038 ] OutputSignal - DEACTIVATED MAIN INC HEATER ON/OFF (-75K1) ';
ARbDeactivateOutput		[38]		:=		DE10205 OR ARbDeactivateTestPB[38];

(*Deactivate*)
ARsDeactivateDescription	[39]		:=		'[ DA-0039 ] OutputSignal - DEACTIVATED RESERVED ';
ARbDeactivateOutput		[39]		:=		DE10206 OR ARbDeactivateTestPB[39];

(*Deactivate*)
ARsDeactivateDescription	[40]		:=		'[ DA-0040 ] OutputSignal - DEACTIVATED RESERVED ';
ARbDeactivateOutput		[40]		:=		DE10207 OR ARbDeactivateTestPB[40];

(*Deactivate*)
ARsDeactivateDescription	[41]		:=		'[ DA-0041 ] OutputSignal - DEACTIVATED RESERVED ';
ARbDeactivateOutput		[41]		:=		DE10208 OR ARbDeactivateTestPB[41];

(*Deactivate*)
ARsDeactivateDescription	[42]		:=		'[ DA-0042 ] OutputSignal - DEACTIVATED RESERVED ';
ARbDeactivateOutput		[42]		:=		DE10209 OR ARbDeactivateTestPB[42];

(*Deactivate*)
ARsDeactivateDescription	[43]		:=		'[ DA-0043 ] OutputSignal - DEACTIVATED RESERVED ';
ARbDeactivateOutput		[43]		:=		DE10210 OR ARbDeactivateTestPB[43];

(*Deactivate*)
ARsDeactivateDescription	[44]		:=		'[ DA-0044 ] OutputSignal - DEACTIVATED RESERVED ';
ARbDeactivateOutput		[44]		:=		DE10211 OR ARbDeactivateTestPB[44];

(*Deactivate*)
ARsDeactivateDescription	[45]		:=		'[ DA-0045 ] OutputSignal - DEACTIVATED RESERVED ';
ARbDeactivateOutput		[45]		:=		DE10212 OR ARbDeactivateTestPB[45];

(*Deactivate*)
ARsDeactivateDescription	[46]		:=		'[ DA-0046 ] OutputSignal - DEACTIVATED RESERVED ';
ARbDeactivateOutput		[46]		:=		DE10213 OR ARbDeactivateTestPB[46];

(*Deactivate*)
ARsDeactivateDescription	[47]		:=		'[ DA-0047 ] OutputSignal - DEACTIVATED RESERVED ';
ARbDeactivateOutput		[47]		:=		DE10214 OR ARbDeactivateTestPB[47];

(*Deactivate*)
ARsDeactivateDescription	[48]		:=		'[ DA-0048 ] OutputSignal - DEACTIVATED RESERVED ';
ARbDeactivateOutput		[48]		:=		DE10215 OR ARbDeactivateTestPB[48];

(********************************************************************************** DEACTIVATED - ( ARbDeactivateOutput[49] - ARbDeactivateOutput[64] )**********************************************************************************)

(*Deactivate*)
ARsDeactivateDescription	[49]		:=		'[ DA-0049 ] OutputSignal - DEACTIVATED RESERVED ';
ARbDeactivateOutput		[49]		:=		FALSE OR ARbDeactivateTestPB[49];

(*Deactivate*)
ARsDeactivateDescription	[50]		:=		'[ DA-0050 ] OutputSignal - DEACTIVATED RESERVED ';
ARbDeactivateOutput		[50]		:=		FALSE OR ARbDeactivateTestPB[50];

(*Deactivate*)
ARsDeactivateDescription	[51]		:=		'[ DA-0051 ] OutputSignal - DEACTIVATED RESERVED ';
ARbDeactivateOutput		[51]		:=		FALSE OR ARbDeactivateTestPB[51];

(*Deactivate*)
ARsDeactivateDescription	[52]		:=		'[ DA-0052 ] OutputSignal - DEACTIVATED RESERVED ';
ARbDeactivateOutput		[52]		:=		FALSE OR ARbDeactivateTestPB[52];

(*Deactivate*)
ARsDeactivateDescription	[53]		:=		'[ DA-0053 ] OutputSignal - DEACTIVATED RESERVED ';
ARbDeactivateOutput		[53]		:=		FALSE OR ARbDeactivateTestPB[53];

(*Deactivate*)
ARsDeactivateDescription	[54]		:=		'[ DA-0054 ] OutputSignal - DEACTIVATED RESERVED ';
ARbDeactivateOutput		[54]		:=		FALSE OR ARbDeactivateTestPB[54];

(*Deactivate*)
ARsDeactivateDescription	[55]		:=		'[ DA-0055 ] OutputSignal - DEACTIVATED RESERVED ';
ARbDeactivateOutput		[55]		:=		FALSE OR ARbDeactivateTestPB[55];

(*Deactivate*)
ARsDeactivateDescription	[56]		:=		'[ DA-0056 ] OutputSignal - DEACTIVATED RESERVED ';
ARbDeactivateOutput		[56]		:=		FALSE OR ARbDeactivateTestPB[56];

(*Deactivate*)
ARsDeactivateDescription	[57]		:=		'[ DA-0057 ] OutputSignal - DEACTIVATED RESERVED ';
ARbDeactivateOutput		[57]		:=		FALSE OR ARbDeactivateTestPB[57];

(*Deactivate*)
ARsDeactivateDescription	[58]		:=		'[ DA-0058 ] OutputSignal - DEACTIVATED RESERVED ';
ARbDeactivateOutput		[58]		:=		FALSE OR ARbDeactivateTestPB[58];

(*Deactivate*)
ARsDeactivateDescription	[59]		:=		'[ DA-0059 ] OutputSignal - DEACTIVATED RESERVED ';
ARbDeactivateOutput		[59]		:=		FALSE OR ARbDeactivateTestPB[59];

(*Deactivate*)
ARsDeactivateDescription	[60]		:=		'[ DA-0060 ] OutputSignal - DEACTIVATED RESERVED ';
ARbDeactivateOutput		[60]		:=		FALSE OR ARbDeactivateTestPB[60];

(*Deactivate*)
ARsDeactivateDescription	[61]		:=		'[ DA-0061 ] OutputSignal - DEACTIVATED RESERVED ';
ARbDeactivateOutput		[61]		:=		FALSE OR ARbDeactivateTestPB[61];

(*Deactivate*)
ARsDeactivateDescription	[62]		:=		'[ DA-0062 ] OutputSignal - DEACTIVATED RESERVED ';
ARbDeactivateOutput		[62]		:=		FALSE OR ARbDeactivateTestPB[62];

(*Deactivate*)
ARsDeactivateDescription	[63]		:=		'[ DA-0063 ] OutputSignal - DEACTIVATED RESERVED ';
ARbDeactivateOutput		[63]		:=		FALSE OR ARbDeactivateTestPB[63];

(*Deactivate*)
ARsDeactivateDescription	[64]		:=		'[ DA-0064 ] OutputSignal - DEACTIVATED RESERVED ';
ARbDeactivateOutput		[64]		:=		FALSE OR ARbDeactivateTestPB[64];

(********************************************************************************** DEACTIVATED - ( ARbDeactivateOutput[65] - ARbDeactivateOutput[80] )**********************************************************************************)

(*Deactivate*)
ARsDeactivateDescription	[65]		:=		'[ DA-0065 ] OutputSignal - DEACTIVATED RESERVED ';
ARbDeactivateOutput		[65]		:=		FALSE OR ARbDeactivateTestPB[65];

(*Deactivate*)
ARsDeactivateDescription	[66]		:=		'[ DA-0066 ] OutputSignal - DEACTIVATED RESERVED ';
ARbDeactivateOutput		[66]		:=		FALSE OR ARbDeactivateTestPB[66];

(*Deactivate*)
ARsDeactivateDescription	[67]		:=		'[ DA-0067 ] OutputSignal - Reserved';
ARbDeactivateOutput		[67]		:=		FALSE OR ARbDeactivateTestPB[67];

(*Deactivate*)
ARsDeactivateDescription	[68]		:=		'[ DA-0068 ] OutputSignal - Reserved';
ARbDeactivateOutput		[68]		:=		FALSE OR ARbDeactivateTestPB[68];

(*Deactivate*)
ARsDeactivateDescription	[69]		:=		'[ DA-0069 ] OutputSignal - Reserved';
ARbDeactivateOutput		[69]		:=		FALSE OR ARbDeactivateTestPB[69];

(*Deactivate*)
ARsDeactivateDescription	[70]		:=		'[ DA-0070 ] OutputSignal - Reserved';
ARbDeactivateOutput		[70]		:=		FALSE OR ARbDeactivateTestPB[70];

(*Deactivate*)
ARsDeactivateDescription	[71]		:=		'[ DA-0071 ] OutputSignal - Reserved';
ARbDeactivateOutput		[71]		:=		FALSE OR ARbDeactivateTestPB[71];

(*Deactivate*)
ARsDeactivateDescription	[72]		:=		'[ DA-0072 ] OutputSignal - Reserved';
ARbDeactivateOutput		[72]		:=		FALSE OR ARbDeactivateTestPB[72];

(*Deactivate*)
ARsDeactivateDescription	[73]		:=		'[ DA-0073 ] OutputSignal - Reserved';
ARbDeactivateOutput		[73]		:=		FALSE OR ARbDeactivateTestPB[73];

(*Deactivate*)
ARsDeactivateDescription	[74]		:=		'[ DA-0074 ] OutputSignal - Reserved';
ARbDeactivateOutput		[74]		:=		FALSE OR ARbDeactivateTestPB[74];

(*Deactivate*)
ARsDeactivateDescription	[75]		:=		'[ DA-0075 ] OutputSignal - Reserved';
ARbDeactivateOutput		[75]		:=		FALSE OR ARbDeactivateTestPB[75];

(*Deactivate*)
ARsDeactivateDescription	[76]		:=		'[ DA-0076 ] OutputSignal - Reserved';
ARbDeactivateOutput		[76]		:=		FALSE OR ARbDeactivateTestPB[76];

(*Deactivate*)
ARsDeactivateDescription	[77]		:=		'[ DA-0077 ] OutputSignal - Reserved';
ARbDeactivateOutput		[77]		:=		FALSE OR ARbDeactivateTestPB[77];

(*Deactivate*)
ARsDeactivateDescription	[78]		:=		'[ DA-0078 ] OutputSignal - Reserved';
ARbDeactivateOutput		[78]		:=		FALSE OR ARbDeactivateTestPB[78];

(*Deactivate*)
ARsDeactivateDescription	[79]		:=		'[ DA-0079 ] OutputSignal - Reserved';
ARbDeactivateOutput		[79]		:=		FALSE OR ARbDeactivateTestPB[79];

(*Deactivate*)
ARsDeactivateDescription	[80]		:=		'[ DA-0080 ] OutputSignal - Alarm Buzzer for Vacuum Disable ';
ARbDeactivateOutput		[80]		:=		bAlarmDeactivated OR ARbDeactivateTestPB[80];

(********************************************************************************** DEACTIVATED - ( ARbDeactivateOutput[81] - ARbDeactivateOutput[96] )**********************************************************************************)

(*Deactivate*)
ARsDeactivateDescription	[81]		:=		'[ DA-0081 ] OutputSignal - Arm 1 MissHook Sensor ByPass 1';
ARbDeactivateOutput		[81]		:=		ARbArmMissHookByPass1[1] OR ARbDeactivateTestPB[81];

(*Deactivate*)
ARsDeactivateDescription	[82]		:=		'[ DA-0082 ] OutputSignal - Arm 1 MissHook Sensor ByPass 2';
ARbDeactivateOutput		[82]		:=		ARbArmMissHookByPass2[1] OR ARbDeactivateTestPB[82];

(*Deactivate*)
ARsDeactivateDescription	[83]		:=		'[ DA-0083 ] OutputSignal - Safety Curtain Sensor Bypass';
ARbDeactivateOutput		[83]		:=		bSafetyDoorSensorBypass OR ARbDeactivateTestPB[83];

(*Deactivate*)
ARsDeactivateDescription	[84]		:=		'[ DA-0084 ] OutputSignal - Arm 1 Crash Sensor ByPass';
ARbDeactivateOutput		[84]		:=		ARbArmCrashByPass[1] OR ARbDeactivateTestPB[84];

(*Deactivate*)
ARsDeactivateDescription	[85]		:=		'[ DA-0085 ] OutputSignal - Conductivity Sensor Bypass';
ARbDeactivateOutput		[85]		:=		ARbConductivityBypass[1] OR ARbDeactivateTestPB[85];

(*Deactivate*)
ARsDeactivateDescription	[86]		:=		'[ DA-0086 ] OutputSignal - Arm 2 MissHook Sensor ByPass 1';
ARbDeactivateOutput		[86]		:=		ARbArmMissHookByPass1[2] OR ARbDeactivateTestPB[86];

(*Deactivate*)
ARsDeactivateDescription	[87]		:=		'[ DA-0087 ] OutputSignal - Arm 2 MissHook Sensor ByPass 2';
ARbDeactivateOutput		[87]		:=		ARbArmMissHookByPass2[2] OR ARbDeactivateTestPB[87];

(*Deactivate*)
ARsDeactivateDescription	[88]		:=		'[ DA-0088 ] OutputSignal - Arm 2 Crash Sensor ByPass';
ARbDeactivateOutput		[88]		:=		ARbArmCrashByPass[2] OR ARbDeactivateTestPB[88];

(*Deactivate*)
ARsDeactivateDescription	[89]		:=		'[ DA-0089 ] OutputSignal - Stn 1 Incoming DI Valve Disable ';
ARbDeactivateOutput		[89]		:=		ARbIncomingDIValveBasedDetergent[1] OR ARbDeactivateTestPB[89];

(*Deactivate*)
ARsDeactivateDescription	[90]		:=		'[ DA-0090 ] OutputSignal - Stn 2 Incoming DI Valve Disable ';
ARbDeactivateOutput		[90]		:=		ARbIncomingDIValveBasedDetergent[2] OR ARbDeactivateTestPB[90];

(*Deactivate*)
ARsDeactivateDescription	[91]		:=		'[ DA-0091 ] OutputSignal - Barcode Function Disable';
ARbDeactivateOutput		[91]		:=		bBarcodeBypass OR ARbDeactivateTestPB[91];

(*Deactivate*)
ARsDeactivateDescription	[92]		:=		'[ DA-0092 ] OutputSignal - Unloading Buzzer Disable ';
ARbDeactivateOutput		[92]		:=		bUnloadingBuzzerDisable OR ARbDeactivateTestPB[92];

(*Deactivate*)
ARsDeactivateDescription	[93]		:=		'[ DA-0093 ] OutputSignal - Station 11 Function Disable ';
ARbDeactivateOutput		[93]		:=		ARbStationFunctionBypass[1] OR ARbDeactivateTestPB[93];

(*Deactivate*)
ARsDeactivateDescription	[94]		:=		'[ DA-0094 ] OutputSignal - Station 12 Function Disable ';
ARbDeactivateOutput		[94]		:=		ARbStationFunctionBypass[2] OR ARbDeactivateTestPB[94];

(*Deactivate*)
ARsDeactivateDescription	[95]		:=		'[ DA-0095 ] OutputSignal - Station 13 Function Disable ';
ARbDeactivateOutput		[95]		:=		ARbStationFunctionBypass[3] OR ARbDeactivateTestPB[95];

(*Deactivate*)
ARsDeactivateDescription	[96]		:=		'[ DA-0096 ] OutputSignal - Station 14 Function Disable ';
ARbDeactivateOutput		[96]		:=		ARbStationFunctionBypass[4] OR ARbDeactivateTestPB[96];

(*Deactivate*)
ARsDeactivateDescription	[97]		:=		'[ DA-0097 ] OutputSignal - Station 15 Function Disable ';
ARbDeactivateOutput		[97]		:=		ARbStationFunctionBypass[5] OR ARbDeactivateTestPB[97];

(*Deactivate*)
ARsDeactivateDescription	[98]		:=		'[ DA-0098 ] OutputSignal - Station 16 Function Disable ';
ARbDeactivateOutput		[98]		:=		ARbStationFunctionBypass[6] OR ARbDeactivateTestPB[98];

(*Deactivate*)
ARsDeactivateDescription	[99]		:=		'[ DA-0099 ] OutputSignal - Station 17 Function Disable ';
ARbDeactivateOutput		[99]		:=		ARbStationFunctionBypass[7] OR ARbDeactivateTestPB[99];

(*Deactivate*)
ARsDeactivateDescription	[100]	:=		'[ DA-0100 ] OutputSignal - Unloading Basket Present - PLEASE IMMEDIATELY UNLOAD THE BASKET ';
ARbDeactivateOutput		[100]	:=		Y100_03 OR ARbDeactivateTestPB[100];
(*
(*Deactivate*)
ARsDeactivateDescription	[101]		:=		'[ DA-0101 ] OutputSignal - Reserved';
ARbDeactivateOutput		[101]		:=		FALSE or ARbDeactivateTestPB[101];

(*Deactivate*)
ARsDeactivateDescription	[102]		:=		'[ DA-0102 ] OutputSignal - Reserved';
ARbDeactivateOutput		[102]		:=		FALSE or ARbDeactivateTestPB[102];

(*Deactivate*)
ARsDeactivateDescription	[103]		:=		'[ DA-0103 ] OutputSignal - Reserved';
ARbDeactivateOutput		[103]		:=		FALSE or ARbDeactivateTestPB[103];

(*Deactivate*)
ARsDeactivateDescription	[104]		:=		'[ DA-0104 ] OutputSignal - Reserved';
ARbDeactivateOutput		[104]		:=		FALSE or ARbDeactivateTestPB[104];

(*Deactivate*)
ARsDeactivateDescription	[105]		:=		'[ DA-0105 ] OutputSignal - Reserved';
ARbDeactivateOutput		[105]		:=		FALSE or ARbDeactivateTestPB[105];

(*Deactivate*)
ARsDeactivateDescription	[106]		:=		'[ DA-0106 ] OutputSignal - Reserved';
ARbDeactivateOutput		[106]		:=		FALSE or ARbDeactivateTestPB[106];

(*Deactivate*)
ARsDeactivateDescription	[107]		:=		'[ DA-0107 ] OutputSignal - Reserved';
ARbDeactivateOutput		[107]		:=		FALSE or ARbDeactivateTestPB[107];

(*Deactivate*)
ARsDeactivateDescription	[108]		:=		'[ DA-0108 ] OutputSignal - Reserved';
ARbDeactivateOutput		[108]		:=		FALSE or ARbDeactivateTestPB[108];

(*Deactivate*)
ARsDeactivateDescription	[109]		:=		'[ DA-0109 ] OutputSignal - Reserved';
ARbDeactivateOutput		[109]		:=		FALSE or ARbDeactivateTestPB[109];

(*Deactivate*)
ARsDeactivateDescription	[110]		:=		'[ DA-0110 ] OutputSignal - Reserved';
ARbDeactivateOutput		[110]		:=		FALSE or ARbDeactivateTestPB[110];

(*Deactivate*)
ARsDeactivateDescription	[111]		:=		'[ DA-0111 ] OutputSignal - Reserved';
ARbDeactivateOutput		[111]		:=		FALSE or ARbDeactivateTestPB[111];

(*Deactivate*)
ARsDeactivateDescription	[112]		:=		'[ DA-0112 ] OutputSignal - Reserved';
ARbDeactivateOutput		[112]		:=		FALSE or ARbDeactivateTestPB[112];

(*Deactivate*)
ARsDeactivateDescription	[113]		:=		'[ DA-0113 ] OutputSignal - Reserved';
ARbDeactivateOutput		[113]		:=		FALSE or ARbDeactivateTestPB[113];

(*Deactivate*)
ARsDeactivateDescription	[114]		:=		'[ DA-0114 ] OutputSignal - Reserved';
ARbDeactivateOutput		[114]		:=		FALSE or ARbDeactivateTestPB[114];

(*Deactivate*)
ARsDeactivateDescription	[115]		:=		'[ DA-0115 ] OutputSignal - Reserved';
ARbDeactivateOutput		[115]		:=		FALSE or ARbDeactivateTestPB[115];

(*Deactivate*)
ARsDeactivateDescription	[116]		:=		'[ DA-0116 ] OutputSignal - Reserved';
ARbDeactivateOutput		[116]		:=		FALSE or ARbDeactivateTestPB[116];

(*Deactivate*)
ARsDeactivateDescription	[117]		:=		'[ DA-0117 ] OutputSignal - Reserved';
ARbDeactivateOutput		[117]		:=		FALSE or ARbDeactivateTestPB[117];

(*Deactivate*)
ARsDeactivateDescription	[118]		:=		'[ DA-0118 ] OutputSignal - Reserved';
ARbDeactivateOutput		[118]		:=		FALSE or ARbDeactivateTestPB[118];

(*Deactivate*)
ARsDeactivateDescription	[119]		:=		'[ DA-0119 ] OutputSignal - Reserved';
ARbDeactivateOutput		[119]		:=		FALSE or ARbDeactivateTestPB[119];

(*Deactivate*)
ARsDeactivateDescription	[120]		:=		'[ DA-0120 ] OutputSignal - Reserved';
ARbDeactivateOutput		[120]		:=		FALSE or ARbDeactivateTestPB[120];

(*Deactivate*)
ARsDeactivateDescription	[121]		:=		'[ DA-0121 ] OutputSignal - Reserved';
ARbDeactivateOutput		[121]		:=		FALSE or ARbDeactivateTestPB[121];

(*Deactivate*)
ARsDeactivateDescription	[122]		:=		'[ DA-0122 ] OutputSignal - Reserved';
ARbDeactivateOutput		[122]		:=		FALSE or ARbDeactivateTestPB[122];

(*Deactivate*)
ARsDeactivateDescription	[123]		:=		'[ DA-0123 ] OutputSignal - Reserved';
ARbDeactivateOutput		[123]		:=		FALSE or ARbDeactivateTestPB[123];

(*Deactivate*)
ARsDeactivateDescription	[124]		:=		'[ DA-0124 ] OutputSignal - Reserved';
ARbDeactivateOutput		[124]		:=		FALSE or ARbDeactivateTestPB[124];

(*Deactivate*)
ARsDeactivateDescription	[125]		:=		'[ DA-0125 ] OutputSignal - Reserved';
ARbDeactivateOutput		[125]		:=		FALSE or ARbDeactivateTestPB[125];

(*Deactivate*)
ARsDeactivateDescription	[126]		:=		'[ DA-0126 ] OutputSignal - Reserved';
ARbDeactivateOutput		[126]		:=		FALSE or ARbDeactivateTestPB[126];

(*Deactivate*)
ARsDeactivateDescription	[127]		:=		'[ DA-0127 ] OutputSignal - Reserved';
ARbDeactivateOutput		[127]		:=		FALSE or ARbDeactivateTestPB[127];

(*Deactivate*)
ARsDeactivateDescription	[128]		:=		'[ DA-0128 ] OutputSignal - Reserved';
ARbDeactivateOutput		[128]		:=		FALSE or ARbDeactivateTestPB[128];

(*Deactivate*)
ARsDeactivateDescription	[129]		:=		'[ DA-0129 ] OutputSignal - Reserved';
ARbDeactivateOutput		[129]		:=		FALSE or ARbDeactivateTestPB[129];

(*Deactivate*)
ARsDeactivateDescription	[130]		:=		'[ DA-0130 ] OutputSignal - Reserved';
ARbDeactivateOutput		[130]		:=		FALSE or ARbDeactivateTestPB[130];

(*Deactivate*)
ARsDeactivateDescription	[131]		:=		'[ DA-0131 ] OutputSignal - Reserved';
ARbDeactivateOutput		[131]		:=		FALSE or ARbDeactivateTestPB[131];

(*Deactivate*)
ARsDeactivateDescription	[132]		:=		'[ DA-0132 ] OutputSignal - Reserved';
ARbDeactivateOutput		[132]		:=		FALSE or ARbDeactivateTestPB[132];

(*Deactivate*)
ARsDeactivateDescription	[133]		:=		'[ DA-0133 ] OutputSignal - Reserved';
ARbDeactivateOutput		[133]		:=		FALSE or ARbDeactivateTestPB[133];

(*Deactivate*)
ARsDeactivateDescription	[134]		:=		'[ DA-0134 ] OutputSignal - Reserved';
ARbDeactivateOutput		[134]		:=		FALSE or ARbDeactivateTestPB[134];

(*Deactivate*)
ARsDeactivateDescription	[135]		:=		'[ DA-0135 ] OutputSignal - Reserved';
ARbDeactivateOutput		[135]		:=		FALSE or ARbDeactivateTestPB[135];

(*Deactivate*)
ARsDeactivateDescription	[136]		:=		'[ DA-0136 ] OutputSignal - Reserved';
ARbDeactivateOutput		[136]		:=		FALSE or ARbDeactivateTestPB[136];

(*Deactivate*)
ARsDeactivateDescription	[137]		:=		'[ DA-0137 ] OutputSignal - Reserved';
ARbDeactivateOutput		[137]		:=		FALSE or ARbDeactivateTestPB[137];

(*Deactivate*)
ARsDeactivateDescription	[138]		:=		'[ DA-0138 ] OutputSignal - Reserved';
ARbDeactivateOutput		[138]		:=		FALSE or ARbDeactivateTestPB[138];

(*Deactivate*)
ARsDeactivateDescription	[139]		:=		'[ DA-0139 ] OutputSignal - Reserved';
ARbDeactivateOutput		[139]		:=		FALSE or ARbDeactivateTestPB[139];

(*Deactivate*)
ARsDeactivateDescription	[140]		:=		'[ DA-0140 ] OutputSignal - Reserved';
ARbDeactivateOutput		[140]		:=		FALSE or ARbDeactivateTestPB[140];

(*Deactivate*)
ARsDeactivateDescription	[141]		:=		'[ DA-0141 ] OutputSignal - Reserved';
ARbDeactivateOutput		[141]		:=		FALSE or ARbDeactivateTestPB[141];

(*Deactivate*)
ARsDeactivateDescription	[142]		:=		'[ DA-0142 ] OutputSignal - Reserved';
ARbDeactivateOutput		[142]		:=		FALSE or ARbDeactivateTestPB[142];

(*Deactivate*)
ARsDeactivateDescription	[143]		:=		'[ DA-0143 ] OutputSignal - Reserved';
ARbDeactivateOutput		[143]		:=		FALSE or ARbDeactivateTestPB[143];

(*Deactivate*)
ARsDeactivateDescription	[144]		:=		'[ DA-0144 ] OutputSignal - Reserved';
ARbDeactivateOutput		[144]		:=		FALSE or ARbDeactivateTestPB[144];

(*Deactivate*)
ARsDeactivateDescription	[145]		:=		'[ DA-0145 ] OutputSignal - Reserved';
ARbDeactivateOutput		[145]		:=		FALSE or ARbDeactivateTestPB[145];

(*Deactivate*)
ARsDeactivateDescription	[146]		:=		'[ DA-0146 ] OutputSignal - Reserved';
ARbDeactivateOutput		[146]		:=		FALSE or ARbDeactivateTestPB[146];

(*Deactivate*)
ARsDeactivateDescription	[147]		:=		'[ DA-0147 ] OutputSignal - Reserved';
ARbDeactivateOutput		[147]		:=		FALSE or ARbDeactivateTestPB[147];

(*Deactivate*)
ARsDeactivateDescription	[148]		:=		'[ DA-0148 ] OutputSignal - Reserved';
ARbDeactivateOutput		[148]		:=		FALSE or ARbDeactivateTestPB[148];

(*Deactivate*)
ARsDeactivateDescription	[149]		:=		'[ DA-0149 ] OutputSignal - Reserved';
ARbDeactivateOutput		[149]		:=		FALSE or ARbDeactivateTestPB[149];

(*Deactivate*)
ARsDeactivateDescription	[150]		:=		'[ DA-0150 ] OutputSignal - Reserved';
ARbDeactivateOutput		[150]		:=		FALSE or ARbDeactivateTestPB[150];

(*Deactivate*)
ARsDeactivateDescription	[151]		:=		'[ DA-0151 ] OutputSignal - Reserved';
ARbDeactivateOutput		[151]		:=		FALSE or ARbDeactivateTestPB[151];

(*Deactivate*)
ARsDeactivateDescription	[152]		:=		'[ DA-0152 ] OutputSignal - Reserved';
ARbDeactivateOutput		[152]		:=		FALSE or ARbDeactivateTestPB[152];

(*Deactivate*)
ARsDeactivateDescription	[153]		:=		'[ DA-0153 ] OutputSignal - Reserved';
ARbDeactivateOutput		[153]		:=		FALSE or ARbDeactivateTestPB[153];

(*Deactivate*)
ARsDeactivateDescription	[154]		:=		'[ DA-0154 ] OutputSignal - Reserved';
ARbDeactivateOutput		[154]		:=		FALSE or ARbDeactivateTestPB[154];

(*Deactivate*)
ARsDeactivateDescription	[155]		:=		'[ DA-0155 ] OutputSignal - Reserved';
ARbDeactivateOutput		[155]		:=		FALSE or ARbDeactivateTestPB[155];

(*Deactivate*)
ARsDeactivateDescription	[156]		:=		'[ DA-0156 ] OutputSignal - Reserved';
ARbDeactivateOutput		[156]		:=		FALSE or ARbDeactivateTestPB[156];

(*Deactivate*)
ARsDeactivateDescription	[157]		:=		'[ DA-0157 ] OutputSignal - Reserved';
ARbDeactivateOutput		[157]		:=		FALSE or ARbDeactivateTestPB[157];

(*Deactivate*)
ARsDeactivateDescription	[158]		:=		'[ DA-0158 ] OutputSignal - Reserved';
ARbDeactivateOutput		[158]		:=		FALSE or ARbDeactivateTestPB[158];

(*Deactivate*)
ARsDeactivateDescription	[159]		:=		'[ DA-0159 ] OutputSignal - Reserved';
ARbDeactivateOutput		[159]		:=		FALSE or ARbDeactivateTestPB[159];

(*Deactivate*)
ARsDeactivateDescription	[160]		:=		'[ DA-0160 ] OutputSignal - Reserved';
ARbDeactivateOutput		[160]		:=		FALSE or ARbDeactivateTestPB[160];

(*Deactivate*)
ARsDeactivateDescription	[161]		:=		'[ DA-0161 ] OutputSignal - Reserved';
ARbDeactivateOutput		[161]		:=		FALSE or ARbDeactivateTestPB[161];

(*Deactivate*)
ARsDeactivateDescription	[162]		:=		'[ DA-0162 ] OutputSignal - Reserved';
ARbDeactivateOutput		[162]		:=		FALSE or ARbDeactivateTestPB[162];

(*Deactivate*)
ARsDeactivateDescription	[163]		:=		'[ DA-0163 ] OutputSignal - Reserved';
ARbDeactivateOutput		[163]		:=		FALSE or ARbDeactivateTestPB[163];

(*Deactivate*)
ARsDeactivateDescription	[164]		:=		'[ DA-0164 ] OutputSignal - Reserved';
ARbDeactivateOutput		[164]		:=		FALSE or ARbDeactivateTestPB[164];

(*Deactivate*)
ARsDeactivateDescription	[165]		:=		'[ DA-0165 ] OutputSignal - Reserved';
ARbDeactivateOutput		[165]		:=		FALSE or ARbDeactivateTestPB[165];

(*Deactivate*)
ARsDeactivateDescription	[166]		:=		'[ DA-0166 ] OutputSignal - Reserved';
ARbDeactivateOutput		[166]		:=		FALSE or ARbDeactivateTestPB[166];

(*Deactivate*)
ARsDeactivateDescription	[167]		:=		'[ DA-0167 ] OutputSignal - Reserved';
ARbDeactivateOutput		[167]		:=		FALSE or ARbDeactivateTestPB[167];

(*Deactivate*)
ARsDeactivateDescription	[168]		:=		'[ DA-0168 ] OutputSignal - Reserved';
ARbDeactivateOutput		[168]		:=		FALSE or ARbDeactivateTestPB[168];

(*Deactivate*)
ARsDeactivateDescription	[169]		:=		'[ DA-0169 ] OutputSignal - Reserved';
ARbDeactivateOutput		[169]		:=		FALSE or ARbDeactivateTestPB[169];

(*Deactivate*)
ARsDeactivateDescription	[170]		:=		'[ DA-0170 ] OutputSignal - Reserved';
ARbDeactivateOutput		[170]		:=		FALSE or ARbDeactivateTestPB[170];

(*Deactivate*)
ARsDeactivateDescription	[171]		:=		'[ DA-0171 ] OutputSignal - Reserved';
ARbDeactivateOutput		[171]		:=		FALSE or ARbDeactivateTestPB[171];

